(* Logix 5000 project; controller IOL_Sample vendor 1 type 14 code 196 rev 30.11; software revision 30.02; part 5 of 7 *)

           TBEN_L4_8IOL:O.Data[90].9   // IO-Link Port 6 - Output data word 8 (INT bit9)
           TBEN_L4_8IOL:O.Data[90].10   // IO-Link Port 6 - Output data word 8 (INT bit10)
           TBEN_L4_8IOL:O.Data[90].11   // IO-Link Port 6 - Output data word 8 (INT bit11)
           TBEN_L4_8IOL:O.Data[90].12   // IO-Link Port 6 - Output data word 8 (INT bit12)
           TBEN_L4_8IOL:O.Data[90].13   // IO-Link Port 6 - Output data word 8 (INT bit13)
           TBEN_L4_8IOL:O.Data[90].14   // IO-Link Port 6 - Output data word 8 (INT bit14)
           TBEN_L4_8IOL:O.Data[90].15   // IO-Link Port 6 - Output data word 8 (INT bit15)
           TBEN_L4_8IOL:O.Data[91]   // IO-Link Port 6 - Output data word 9
           TBEN_L4_8IOL:O.Data[91].0   // IO-Link Port 6 - Output data word 9 (INT bit0)
           TBEN_L4_8IOL:O.Data[91].1   // IO-Link Port 6 - Output data word 9 (INT bit1)
           TBEN_L4_8IOL:O.Data[91].2   // IO-Link Port 6 - Output data word 9 (INT bit2)
           TBEN_L4_8IOL:O.Data[91].3   // IO-Link Port 6 - Output data word 9 (INT bit3)
           TBEN_L4_8IOL:O.Data[91].4   // IO-Link Port 6 - Output data word 9 (INT bit4)
           TBEN_L4_8IOL:O.Data[91].5   // IO-Link Port 6 - Output data word 9 (INT bit5)
           TBEN_L4_8IOL:O.Data[91].6   // IO-Link Port 6 - Output data word 9 (INT bit6)
           TBEN_L4_8IOL:O.Data[91].7   // IO-Link Port 6 - Output data word 9 (INT bit7)
           TBEN_L4_8IOL:O.Data[91].8   // IO-Link Port 6 - Output data word 9 (INT bit8)
           TBEN_L4_8IOL:O.Data[91].9   // IO-Link Port 6 - Output data word 9 (INT bit9)
           TBEN_L4_8IOL:O.Data[91].10   // IO-Link Port 6 - Output data word 9 (INT bit10)
           TBEN_L4_8IOL:O.Data[91].11   // IO-Link Port 6 - Output data word 9 (INT bit11)
           TBEN_L4_8IOL:O.Data[91].12   // IO-Link Port 6 - Output data word 9 (INT bit12)
           TBEN_L4_8IOL:O.Data[91].13   // IO-Link Port 6 - Output data word 9 (INT bit13)
           TBEN_L4_8IOL:O.Data[91].14   // IO-Link Port 6 - Output data word 9 (INT bit14)
           TBEN_L4_8IOL:O.Data[91].15   // IO-Link Port 6 - Output data word 9 (INT bit15)
           TBEN_L4_8IOL:O.Data[92]   // IO-Link Port 6 - Output data word 10
           TBEN_L4_8IOL:O.Data[92].0   // IO-Link Port 6 - Output data word 10 (INT bit0)
           TBEN_L4_8IOL:O.Data[92].1   // IO-Link Port 6 - Output data word 10 (INT bit1)
           TBEN_L4_8IOL:O.Data[92].2   // IO-Link Port 6 - Output data word 10 (INT bit2)
           TBEN_L4_8IOL:O.Data[92].3   // IO-Link Port 6 - Output data word 10 (INT bit3)
           TBEN_L4_8IOL:O.Data[92].4   // IO-Link Port 6 - Output data word 10 (INT bit4)
           TBEN_L4_8IOL:O.Data[92].5   // IO-Link Port 6 - Output data word 10 (INT bit5)
           TBEN_L4_8IOL:O.Data[92].6   // IO-Link Port 6 - Output data word 10 (INT bit6)
           TBEN_L4_8IOL:O.Data[92].7   // IO-Link Port 6 - Output data word 10 (INT bit7)
           TBEN_L4_8IOL:O.Data[92].8   // IO-Link Port 6 - Output data word 10 (INT bit8)
           TBEN_L4_8IOL:O.Data[92].9   // IO-Link Port 6 - Output data word 10 (INT bit9)
           TBEN_L4_8IOL:O.Data[92].10   // IO-Link Port 6 - Output data word 10 (INT bit10)
           TBEN_L4_8IOL:O.Data[92].11   // IO-Link Port 6 - Output data word 10 (INT bit11)
           TBEN_L4_8IOL:O.Data[92].12   // IO-Link Port 6 - Output data word 10 (INT bit12)
           TBEN_L4_8IOL:O.Data[92].13   // IO-Link Port 6 - Output data word 10 (INT bit13)
           TBEN_L4_8IOL:O.Data[92].14   // IO-Link Port 6 - Output data word 10 (INT bit14)
           TBEN_L4_8IOL:O.Data[92].15   // IO-Link Port 6 - Output data word 10 (INT bit15)
           TBEN_L4_8IOL:O.Data[93]   // IO-Link Port 6 - Output data word 11
           TBEN_L4_8IOL:O.Data[93].0   // IO-Link Port 6 - Output data word 11 (INT bit0)
           TBEN_L4_8IOL:O.Data[93].1   // IO-Link Port 6 - Output data word 11 (INT bit1)
           TBEN_L4_8IOL:O.Data[93].2   // IO-Link Port 6 - Output data word 11 (INT bit2)
           TBEN_L4_8IOL:O.Data[93].3   // IO-Link Port 6 - Output data word 11 (INT bit3)
           TBEN_L4_8IOL:O.Data[93].4   // IO-Link Port 6 - Output data word 11 (INT bit4)
           TBEN_L4_8IOL:O.Data[93].5   // IO-Link Port 6 - Output data word 11 (INT bit5)
           TBEN_L4_8IOL:O.Data[93].6   // IO-Link Port 6 - Output data word 11 (INT bit6)
           TBEN_L4_8IOL:O.Data[93].7   // IO-Link Port 6 - Output data word 11 (INT bit7)
           TBEN_L4_8IOL:O.Data[93].8   // IO-Link Port 6 - Output data word 11 (INT bit8)
           TBEN_L4_8IOL:O.Data[93].9   // IO-Link Port 6 - Output data word 11 (INT bit9)
           TBEN_L4_8IOL:O.Data[93].10   // IO-Link Port 6 - Output data word 11 (INT bit10)
           TBEN_L4_8IOL:O.Data[93].11   // IO-Link Port 6 - Output data word 11 (INT bit11)
           TBEN_L4_8IOL:O.Data[93].12   // IO-Link Port 6 - Output data word 11 (INT bit12)
           TBEN_L4_8IOL:O.Data[93].13   // IO-Link Port 6 - Output data word 11 (INT bit13)
           TBEN_L4_8IOL:O.Data[93].14   // IO-Link Port 6 - Output data word 11 (INT bit14)
           TBEN_L4_8IOL:O.Data[93].15   // IO-Link Port 6 - Output data word 11 (INT bit15)
           TBEN_L4_8IOL:O.Data[94]   // IO-Link Port 6 - Output data word 12
           TBEN_L4_8IOL:O.Data[94].0   // IO-Link Port 6 - Output data word 12 (INT bit0)
           TBEN_L4_8IOL:O.Data[94].1   // IO-Link Port 6 - Output data word 12 (INT bit1)
           TBEN_L4_8IOL:O.Data[94].2   // IO-Link Port 6 - Output data word 12 (INT bit2)
           TBEN_L4_8IOL:O.Data[94].3   // IO-Link Port 6 - Output data word 12 (INT bit3)
           TBEN_L4_8IOL:O.Data[94].4   // IO-Link Port 6 - Output data word 12 (INT bit4)
           TBEN_L4_8IOL:O.Data[94].5   // IO-Link Port 6 - Output data word 12 (INT bit5)
           TBEN_L4_8IOL:O.Data[94].6   // IO-Link Port 6 - Output data word 12 (INT bit6)
           TBEN_L4_8IOL:O.Data[94].7   // IO-Link Port 6 - Output data word 12 (INT bit7)
           TBEN_L4_8IOL:O.Data[94].8   // IO-Link Port 6 - Output data word 12 (INT bit8)
           TBEN_L4_8IOL:O.Data[94].9   // IO-Link Port 6 - Output data word 12 (INT bit9)
           TBEN_L4_8IOL:O.Data[94].10   // IO-Link Port 6 - Output data word 12 (INT bit10)
           TBEN_L4_8IOL:O.Data[94].11   // IO-Link Port 6 - Output data word 12 (INT bit11)
           TBEN_L4_8IOL:O.Data[94].12   // IO-Link Port 6 - Output data word 12 (INT bit12)
           TBEN_L4_8IOL:O.Data[94].13   // IO-Link Port 6 - Output data word 12 (INT bit13)
           TBEN_L4_8IOL:O.Data[94].14   // IO-Link Port 6 - Output data word 12 (INT bit14)
           TBEN_L4_8IOL:O.Data[94].15   // IO-Link Port 6 - Output data word 12 (INT bit15)
           TBEN_L4_8IOL:O.Data[95]   // IO-Link Port 6 - Output data word 13
           TBEN_L4_8IOL:O.Data[95].0   // IO-Link Port 6 - Output data word 13 (INT bit0)
           TBEN_L4_8IOL:O.Data[95].1   // IO-Link Port 6 - Output data word 13 (INT bit1)
           TBEN_L4_8IOL:O.Data[95].2   // IO-Link Port 6 - Output data word 13 (INT bit2)
           TBEN_L4_8IOL:O.Data[95].3   // IO-Link Port 6 - Output data word 13 (INT bit3)
           TBEN_L4_8IOL:O.Data[95].4   // IO-Link Port 6 - Output data word 13 (INT bit4)
           TBEN_L4_8IOL:O.Data[95].5   // IO-Link Port 6 - Output data word 13 (INT bit5)
           TBEN_L4_8IOL:O.Data[95].6   // IO-Link Port 6 - Output data word 13 (INT bit6)
           TBEN_L4_8IOL:O.Data[95].7   // IO-Link Port 6 - Output data word 13 (INT bit7)
           TBEN_L4_8IOL:O.Data[95].8   // IO-Link Port 6 - Output data word 13 (INT bit8)
           TBEN_L4_8IOL:O.Data[95].9   // IO-Link Port 6 - Output data word 13 (INT bit9)
           TBEN_L4_8IOL:O.Data[95].10   // IO-Link Port 6 - Output data word 13 (INT bit10)
           TBEN_L4_8IOL:O.Data[95].11   // IO-Link Port 6 - Output data word 13 (INT bit11)
           TBEN_L4_8IOL:O.Data[95].12   // IO-Link Port 6 - Output data word 13 (INT bit12)
           TBEN_L4_8IOL:O.Data[95].13   // IO-Link Port 6 - Output data word 13 (INT bit13)
           TBEN_L4_8IOL:O.Data[95].14   // IO-Link Port 6 - Output data word 13 (INT bit14)
           TBEN_L4_8IOL:O.Data[95].15   // IO-Link Port 6 - Output data word 13 (INT bit15)
           TBEN_L4_8IOL:O.Data[96]   // IO-Link Port 6 - Output data word 14
           TBEN_L4_8IOL:O.Data[96].0   // IO-Link Port 6 - Output data word 14 (INT bit0)
           TBEN_L4_8IOL:O.Data[96].1   // IO-Link Port 6 - Output data word 14 (INT bit1)
           TBEN_L4_8IOL:O.Data[96].2   // IO-Link Port 6 - Output data word 14 (INT bit2)
           TBEN_L4_8IOL:O.Data[96].3   // IO-Link Port 6 - Output data word 14 (INT bit3)
           TBEN_L4_8IOL:O.Data[96].4   // IO-Link Port 6 - Output data word 14 (INT bit4)
           TBEN_L4_8IOL:O.Data[96].5   // IO-Link Port 6 - Output data word 14 (INT bit5)
           TBEN_L4_8IOL:O.Data[96].6   // IO-Link Port 6 - Output data word 14 (INT bit6)
           TBEN_L4_8IOL:O.Data[96].7   // IO-Link Port 6 - Output data word 14 (INT bit7)
           TBEN_L4_8IOL:O.Data[96].8   // IO-Link Port 6 - Output data word 14 (INT bit8)
           TBEN_L4_8IOL:O.Data[96].9   // IO-Link Port 6 - Output data word 14 (INT bit9)
           TBEN_L4_8IOL:O.Data[96].10   // IO-Link Port 6 - Output data word 14 (INT bit10)
           TBEN_L4_8IOL:O.Data[96].11   // IO-Link Port 6 - Output data word 14 (INT bit11)
           TBEN_L4_8IOL:O.Data[96].12   // IO-Link Port 6 - Output data word 14 (INT bit12)
           TBEN_L4_8IOL:O.Data[96].13   // IO-Link Port 6 - Output data word 14 (INT bit13)
           TBEN_L4_8IOL:O.Data[96].14   // IO-Link Port 6 - Output data word 14 (INT bit14)
           TBEN_L4_8IOL:O.Data[96].15   // IO-Link Port 6 - Output data word 14 (INT bit15)
           TBEN_L4_8IOL:O.Data[97]   // IO-Link Port 6 - Output data word 15
           TBEN_L4_8IOL:O.Data[97].0   // IO-Link Port 6 - Output data word 15 (INT bit0)
           TBEN_L4_8IOL:O.Data[97].1   // IO-Link Port 6 - Output data word 15 (INT bit1)
           TBEN_L4_8IOL:O.Data[97].2   // IO-Link Port 6 - Output data word 15 (INT bit2)
           TBEN_L4_8IOL:O.Data[97].3   // IO-Link Port 6 - Output data word 15 (INT bit3)
           TBEN_L4_8IOL:O.Data[97].4   // IO-Link Port 6 - Output data word 15 (INT bit4)
           TBEN_L4_8IOL:O.Data[97].5   // IO-Link Port 6 - Output data word 15 (INT bit5)
           TBEN_L4_8IOL:O.Data[97].6   // IO-Link Port 6 - Output data word 15 (INT bit6)
           TBEN_L4_8IOL:O.Data[97].7   // IO-Link Port 6 - Output data word 15 (INT bit7)
           TBEN_L4_8IOL:O.Data[97].8   // IO-Link Port 6 - Output data word 15 (INT bit8)
           TBEN_L4_8IOL:O.Data[97].9   // IO-Link Port 6 - Output data word 15 (INT bit9)
           TBEN_L4_8IOL:O.Data[97].10   // IO-Link Port 6 - Output data word 15 (INT bit10)
           TBEN_L4_8IOL:O.Data[97].11   // IO-Link Port 6 - Output data word 15 (INT bit11)
           TBEN_L4_8IOL:O.Data[97].12   // IO-Link Port 6 - Output data word 15 (INT bit12)
           TBEN_L4_8IOL:O.Data[97].13   // IO-Link Port 6 - Output data word 15 (INT bit13)
           TBEN_L4_8IOL:O.Data[97].14   // IO-Link Port 6 - Output data word 15 (INT bit14)
           TBEN_L4_8IOL:O.Data[97].15   // IO-Link Port 6 - Output data word 15 (INT bit15)
           TBEN_L4_8IOL:O.Data[98]   // IO-Link Port 7 - Output data word 0
           TBEN_L4_8IOL:O.Data[98].0   // IO-Link Port 7 - Output data word 0 (INT bit0)
           TBEN_L4_8IOL:O.Data[98].1   // IO-Link Port 7 - Output data word 0 (INT bit1)
           TBEN_L4_8IOL:O.Data[98].2   // IO-Link Port 7 - Output data word 0 (INT bit2)
           TBEN_L4_8IOL:O.Data[98].3   // IO-Link Port 7 - Output data word 0 (INT bit3)
           TBEN_L4_8IOL:O.Data[98].4   // IO-Link Port 7 - Output data word 0 (INT bit4)
           TBEN_L4_8IOL:O.Data[98].5   // IO-Link Port 7 - Output data word 0 (INT bit5)
           TBEN_L4_8IOL:O.Data[98].6   // IO-Link Port 7 - Output data word 0 (INT bit6)
           TBEN_L4_8IOL:O.Data[98].7   // IO-Link Port 7 - Output data word 0 (INT bit7)
           TBEN_L4_8IOL:O.Data[98].8   // IO-Link Port 7 - Output data word 0 (INT bit8)
           TBEN_L4_8IOL:O.Data[98].9   // IO-Link Port 7 - Output data word 0 (INT bit9)
           TBEN_L4_8IOL:O.Data[98].10   // IO-Link Port 7 - Output data word 0 (INT bit10)
           TBEN_L4_8IOL:O.Data[98].11   // IO-Link Port 7 - Output data word 0 (INT bit11)
           TBEN_L4_8IOL:O.Data[98].12   // IO-Link Port 7 - Output data word 0 (INT bit12)
           TBEN_L4_8IOL:O.Data[98].13   // IO-Link Port 7 - Output data word 0 (INT bit13)
           TBEN_L4_8IOL:O.Data[98].14   // IO-Link Port 7 - Output data word 0 (INT bit14)
           TBEN_L4_8IOL:O.Data[98].15   // IO-Link Port 7 - Output data word 0 (INT bit15)
           TBEN_L4_8IOL:O.Data[99]   // IO-Link Port 7 - Output data word 1
           TBEN_L4_8IOL:O.Data[99].0   // IO-Link Port 7 - Output data word 1 (INT bit0)
           TBEN_L4_8IOL:O.Data[99].1   // IO-Link Port 7 - Output data word 1 (INT bit1)
           TBEN_L4_8IOL:O.Data[99].2   // IO-Link Port 7 - Output data word 1 (INT bit2)
           TBEN_L4_8IOL:O.Data[99].3   // IO-Link Port 7 - Output data word 1 (INT bit3)
           TBEN_L4_8IOL:O.Data[99].4   // IO-Link Port 7 - Output data word 1 (INT bit4)
           TBEN_L4_8IOL:O.Data[99].5   // IO-Link Port 7 - Output data word 1 (INT bit5)
           TBEN_L4_8IOL:O.Data[99].6   // IO-Link Port 7 - Output data word 1 (INT bit6)
           TBEN_L4_8IOL:O.Data[99].7   // IO-Link Port 7 - Output data word 1 (INT bit7)
           TBEN_L4_8IOL:O.Data[99].8   // IO-Link Port 7 - Output data word 1 (INT bit8)
           TBEN_L4_8IOL:O.Data[99].9   // IO-Link Port 7 - Output data word 1 (INT bit9)
           TBEN_L4_8IOL:O.Data[99].10   // IO-Link Port 7 - Output data word 1 (INT bit10)
           TBEN_L4_8IOL:O.Data[99].11   // IO-Link Port 7 - Output data word 1 (INT bit11)
           TBEN_L4_8IOL:O.Data[99].12   // IO-Link Port 7 - Output data word 1 (INT bit12)
           TBEN_L4_8IOL:O.Data[99].13   // IO-Link Port 7 - Output data word 1 (INT bit13)
           TBEN_L4_8IOL:O.Data[99].14   // IO-Link Port 7 - Output data word 1 (INT bit14)
           TBEN_L4_8IOL:O.Data[99].15   // IO-Link Port 7 - Output data word 1 (INT bit15)
           TBEN_L4_8IOL:O.Data[100]   // IO-Link Port 7 - Output data word 2
           TBEN_L4_8IOL:O.Data[100].0   // IO-Link Port 7 - Output data word 2 (INT bit0)
           TBEN_L4_8IOL:O.Data[100].1   // IO-Link Port 7 - Output data word 2 (INT bit1)
           TBEN_L4_8IOL:O.Data[100].2   // IO-Link Port 7 - Output data word 2 (INT bit2)
           TBEN_L4_8IOL:O.Data[100].3   // IO-Link Port 7 - Output data word 2 (INT bit3)
           TBEN_L4_8IOL:O.Data[100].4   // IO-Link Port 7 - Output data word 2 (INT bit4)
           TBEN_L4_8IOL:O.Data[100].5   // IO-Link Port 7 - Output data word 2 (INT bit5)
           TBEN_L4_8IOL:O.Data[100].6   // IO-Link Port 7 - Output data word 2 (INT bit6)
           TBEN_L4_8IOL:O.Data[100].7   // IO-Link Port 7 - Output data word 2 (INT bit7)
           TBEN_L4_8IOL:O.Data[100].8   // IO-Link Port 7 - Output data word 2 (INT bit8)
           TBEN_L4_8IOL:O.Data[100].9   // IO-Link Port 7 - Output data word 2 (INT bit9)
           TBEN_L4_8IOL:O.Data[100].10   // IO-Link Port 7 - Output data word 2 (INT bit10)
           TBEN_L4_8IOL:O.Data[100].11   // IO-Link Port 7 - Output data word 2 (INT bit11)
           TBEN_L4_8IOL:O.Data[100].12   // IO-Link Port 7 - Output data word 2 (INT bit12)
           TBEN_L4_8IOL:O.Data[100].13   // IO-Link Port 7 - Output data word 2 (INT bit13)
           TBEN_L4_8IOL:O.Data[100].14   // IO-Link Port 7 - Output data word 2 (INT bit14)
           TBEN_L4_8IOL:O.Data[100].15   // IO-Link Port 7 - Output data word 2 (INT bit15)
           TBEN_L4_8IOL:O.Data[101]   // IO-Link Port 7 - Output data word 3
           TBEN_L4_8IOL:O.Data[101].0   // IO-Link Port 7 - Output data word 3 (INT bit0)
           TBEN_L4_8IOL:O.Data[101].1   // IO-Link Port 7 - Output data word 3 (INT bit1)
           TBEN_L4_8IOL:O.Data[101].2   // IO-Link Port 7 - Output data word 3 (INT bit2)
           TBEN_L4_8IOL:O.Data[101].3   // IO-Link Port 7 - Output data word 3 (INT bit3)
           TBEN_L4_8IOL:O.Data[101].4   // IO-Link Port 7 - Output data word 3 (INT bit4)
           TBEN_L4_8IOL:O.Data[101].5   // IO-Link Port 7 - Output data word 3 (INT bit5)
           TBEN_L4_8IOL:O.Data[101].6   // IO-Link Port 7 - Output data word 3 (INT bit6)
           TBEN_L4_8IOL:O.Data[101].7   // IO-Link Port 7 - Output data word 3 (INT bit7)
           TBEN_L4_8IOL:O.Data[101].8   // IO-Link Port 7 - Output data word 3 (INT bit8)
           TBEN_L4_8IOL:O.Data[101].9   // IO-Link Port 7 - Output data word 3 (INT bit9)
           TBEN_L4_8IOL:O.Data[101].10   // IO-Link Port 7 - Output data word 3 (INT bit10)
           TBEN_L4_8IOL:O.Data[101].11   // IO-Link Port 7 - Output data word 3 (INT bit11)
           TBEN_L4_8IOL:O.Data[101].12   // IO-Link Port 7 - Output data word 3 (INT bit12)
           TBEN_L4_8IOL:O.Data[101].13   // IO-Link Port 7 - Output data word 3 (INT bit13)
           TBEN_L4_8IOL:O.Data[101].14   // IO-Link Port 7 - Output data word 3 (INT bit14)
           TBEN_L4_8IOL:O.Data[101].15   // IO-Link Port 7 - Output data word 3 (INT bit15)
           TBEN_L4_8IOL:O.Data[102]   // IO-Link Port 7 - Output data word 4
           TBEN_L4_8IOL:O.Data[102].0   // IO-Link Port 7 - Output data word 4 (INT bit0)
           TBEN_L4_8IOL:O.Data[102].1   // IO-Link Port 7 - Output data word 4 (INT bit1)
           TBEN_L4_8IOL:O.Data[102].2   // IO-Link Port 7 - Output data word 4 (INT bit2)
           TBEN_L4_8IOL:O.Data[102].3   // IO-Link Port 7 - Output data word 4 (INT bit3)
           TBEN_L4_8IOL:O.Data[102].4   // IO-Link Port 7 - Output data word 4 (INT bit4)
           TBEN_L4_8IOL:O.Data[102].5   // IO-Link Port 7 - Output data word 4 (INT bit5)
           TBEN_L4_8IOL:O.Data[102].6   // IO-Link Port 7 - Output data word 4 (INT bit6)
           TBEN_L4_8IOL:O.Data[102].7   // IO-Link Port 7 - Output data word 4 (INT bit7)
           TBEN_L4_8IOL:O.Data[102].8   // IO-Link Port 7 - Output data word 4 (INT bit8)
           TBEN_L4_8IOL:O.Data[102].9   // IO-Link Port 7 - Output data word 4 (INT bit9)
           TBEN_L4_8IOL:O.Data[102].10   // IO-Link Port 7 - Output data word 4 (INT bit10)
           TBEN_L4_8IOL:O.Data[102].11   // IO-Link Port 7 - Output data word 4 (INT bit11)
           TBEN_L4_8IOL:O.Data[102].12   // IO-Link Port 7 - Output data word 4 (INT bit12)
           TBEN_L4_8IOL:O.Data[102].13   // IO-Link Port 7 - Output data word 4 (INT bit13)
           TBEN_L4_8IOL:O.Data[102].14   // IO-Link Port 7 - Output data word 4 (INT bit14)
           TBEN_L4_8IOL:O.Data[102].15   // IO-Link Port 7 - Output data word 4 (INT bit15)
           TBEN_L4_8IOL:O.Data[103]   // IO-Link Port 7 - Output data word 5
           TBEN_L4_8IOL:O.Data[103].0   // IO-Link Port 7 - Output data word 5 (INT bit0)
           TBEN_L4_8IOL:O.Data[103].1   // IO-Link Port 7 - Output data word 5 (INT bit1)
           TBEN_L4_8IOL:O.Data[103].2   // IO-Link Port 7 - Output data word 5 (INT bit2)
           TBEN_L4_8IOL:O.Data[103].3   // IO-Link Port 7 - Output data word 5 (INT bit3)
           TBEN_L4_8IOL:O.Data[103].4   // IO-Link Port 7 - Output data word 5 (INT bit4)
           TBEN_L4_8IOL:O.Data[103].5   // IO-Link Port 7 - Output data word 5 (INT bit5)
           TBEN_L4_8IOL:O.Data[103].6   // IO-Link Port 7 - Output data word 5 (INT bit6)
           TBEN_L4_8IOL:O.Data[103].7   // IO-Link Port 7 - Output data word 5 (INT bit7)
           TBEN_L4_8IOL:O.Data[103].8   // IO-Link Port 7 - Output data word 5 (INT bit8)
           TBEN_L4_8IOL:O.Data[103].9   // IO-Link Port 7 - Output data word 5 (INT bit9)
           TBEN_L4_8IOL:O.Data[103].10   // IO-Link Port 7 - Output data word 5 (INT bit10)
           TBEN_L4_8IOL:O.Data[103].11   // IO-Link Port 7 - Output data word 5 (INT bit11)
           TBEN_L4_8IOL:O.Data[103].12   // IO-Link Port 7 - Output data word 5 (INT bit12)
           TBEN_L4_8IOL:O.Data[103].13   // IO-Link Port 7 - Output data word 5 (INT bit13)
           TBEN_L4_8IOL:O.Data[103].14   // IO-Link Port 7 - Output data word 5 (INT bit14)
           TBEN_L4_8IOL:O.Data[103].15   // IO-Link Port 7 - Output data word 5 (INT bit15)
           TBEN_L4_8IOL:O.Data[104]   // IO-Link Port 7 - Output data word 6
           TBEN_L4_8IOL:O.Data[104].0   // IO-Link Port 7 - Output data word 6 (INT bit0)
           TBEN_L4_8IOL:O.Data[104].1   // IO-Link Port 7 - Output data word 6 (INT bit1)
           TBEN_L4_8IOL:O.Data[104].2   // IO-Link Port 7 - Output data word 6 (INT bit2)
           TBEN_L4_8IOL:O.Data[104].3   // IO-Link Port 7 - Output data word 6 (INT bit3)
           TBEN_L4_8IOL:O.Data[104].4   // IO-Link Port 7 - Output data word 6 (INT bit4)
           TBEN_L4_8IOL:O.Data[104].5   // IO-Link Port 7 - Output data word 6 (INT bit5)
           TBEN_L4_8IOL:O.Data[104].6   // IO-Link Port 7 - Output data word 6 (INT bit6)
           TBEN_L4_8IOL:O.Data[104].7   // IO-Link Port 7 - Output data word 6 (INT bit7)
           TBEN_L4_8IOL:O.Data[104].8   // IO-Link Port 7 - Output data word 6 (INT bit8)
           TBEN_L4_8IOL:O.Data[104].9   // IO-Link Port 7 - Output data word 6 (INT bit9)
           TBEN_L4_8IOL:O.Data[104].10   // IO-Link Port 7 - Output data word 6 (INT bit10)
           TBEN_L4_8IOL:O.Data[104].11   // IO-Link Port 7 - Output data word 6 (INT bit11)
           TBEN_L4_8IOL:O.Data[104].12   // IO-Link Port 7 - Output data word 6 (INT bit12)
           TBEN_L4_8IOL:O.Data[104].13   // IO-Link Port 7 - Output data word 6 (INT bit13)
           TBEN_L4_8IOL:O.Data[104].14   // IO-Link Port 7 - Output data word 6 (INT bit14)
           TBEN_L4_8IOL:O.Data[104].15   // IO-Link Port 7 - Output data word 6 (INT bit15)
           TBEN_L4_8IOL:O.Data[105]   // IO-Link Port 7 - Output data word 7
           TBEN_L4_8IOL:O.Data[105].0   // IO-Link Port 7 - Output data word 7 (INT bit0)
           TBEN_L4_8IOL:O.Data[105].1   // IO-Link Port 7 - Output data word 7 (INT bit1)
           TBEN_L4_8IOL:O.Data[105].2   // IO-Link Port 7 - Output data word 7 (INT bit2)
           TBEN_L4_8IOL:O.Data[105].3   // IO-Link Port 7 - Output data word 7 (INT bit3)
           TBEN_L4_8IOL:O.Data[105].4   // IO-Link Port 7 - Output data word 7 (INT bit4)
           TBEN_L4_8IOL:O.Data[105].5   // IO-Link Port 7 - Output data word 7 (INT bit5)
           TBEN_L4_8IOL:O.Data[105].6   // IO-Link Port 7 - Output data word 7 (INT bit6)
           TBEN_L4_8IOL:O.Data[105].7   // IO-Link Port 7 - Output data word 7 (INT bit7)
           TBEN_L4_8IOL:O.Data[105].8   // IO-Link Port 7 - Output data word 7 (INT bit8)
           TBEN_L4_8IOL:O.Data[105].9   // IO-Link Port 7 - Output data word 7 (INT bit9)
           TBEN_L4_8IOL:O.Data[105].10   // IO-Link Port 7 - Output data word 7 (INT bit10)
           TBEN_L4_8IOL:O.Data[105].11   // IO-Link Port 7 - Output data word 7 (INT bit11)
           TBEN_L4_8IOL:O.Data[105].12   // IO-Link Port 7 - Output data word 7 (INT bit12)
           TBEN_L4_8IOL:O.Data[105].13   // IO-Link Port 7 - Output data word 7 (INT bit13)
           TBEN_L4_8IOL:O.Data[105].14   // IO-Link Port 7 - Output data word 7 (INT bit14)
           TBEN_L4_8IOL:O.Data[105].15   // IO-Link Port 7 - Output data word 7 (INT bit15)
           TBEN_L4_8IOL:O.Data[106]   // IO-Link Port 7 - Output data word 8
           TBEN_L4_8IOL:O.Data[106].0   // IO-Link Port 7 - Output data word 8 (INT bit0)
           TBEN_L4_8IOL:O.Data[106].1   // IO-Link Port 7 - Output data word 8 (INT bit1)
           TBEN_L4_8IOL:O.Data[106].2   // IO-Link Port 7 - Output data word 8 (INT bit2)
           TBEN_L4_8IOL:O.Data[106].3   // IO-Link Port 7 - Output data word 8 (INT bit3)
           TBEN_L4_8IOL:O.Data[106].4   // IO-Link Port 7 - Output data word 8 (INT bit4)
           TBEN_L4_8IOL:O.Data[106].5   // IO-Link Port 7 - Output data word 8 (INT bit5)
           TBEN_L4_8IOL:O.Data[106].6   // IO-Link Port 7 - Output data word 8 (INT bit6)
           TBEN_L4_8IOL:O.Data[106].7   // IO-Link Port 7 - Output data word 8 (INT bit7)
           TBEN_L4_8IOL:O.Data[106].8   // IO-Link Port 7 - Output data word 8 (INT bit8)
           TBEN_L4_8IOL:O.Data[106].9   // IO-Link Port 7 - Output data word 8 (INT bit9)
           TBEN_L4_8IOL:O.Data[106].10   // IO-Link Port 7 - Output data word 8 (INT bit10)
           TBEN_L4_8IOL:O.Data[106].11   // IO-Link Port 7 - Output data word 8 (INT bit11)
           TBEN_L4_8IOL:O.Data[106].12   // IO-Link Port 7 - Output data word 8 (INT bit12)
           TBEN_L4_8IOL:O.Data[106].13   // IO-Link Port 7 - Output data word 8 (INT bit13)
           TBEN_L4_8IOL:O.Data[106].14   // IO-Link Port 7 - Output data word 8 (INT bit14)
           TBEN_L4_8IOL:O.Data[106].15   // IO-Link Port 7 - Output data word 8 (INT bit15)
           TBEN_L4_8IOL:O.Data[107]   // IO-Link Port 7 - Output data word 9
           TBEN_L4_8IOL:O.Data[107].0   // IO-Link Port 7 - Output data word 9 (INT bit0)
           TBEN_L4_8IOL:O.Data[107].1   // IO-Link Port 7 - Output data word 9 (INT bit1)
           TBEN_L4_8IOL:O.Data[107].2   // IO-Link Port 7 - Output data word 9 (INT bit2)
           TBEN_L4_8IOL:O.Data[107].3   // IO-Link Port 7 - Output data word 9 (INT bit3)
           TBEN_L4_8IOL:O.Data[107].4   // IO-Link Port 7 - Output data word 9 (INT bit4)
           TBEN_L4_8IOL:O.Data[107].5   // IO-Link Port 7 - Output data word 9 (INT bit5)
           TBEN_L4_8IOL:O.Data[107].6   // IO-Link Port 7 - Output data word 9 (INT bit6)
           TBEN_L4_8IOL:O.Data[107].7   // IO-Link Port 7 - Output data word 9 (INT bit7)
           TBEN_L4_8IOL:O.Data[107].8   // IO-Link Port 7 - Output data word 9 (INT bit8)
           TBEN_L4_8IOL:O.Data[107].9   // IO-Link Port 7 - Output data word 9 (INT bit9)
           TBEN_L4_8IOL:O.Data[107].10   // IO-Link Port 7 - Output data word 9 (INT bit10)
           TBEN_L4_8IOL:O.Data[107].11   // IO-Link Port 7 - Output data word 9 (INT bit11)
           TBEN_L4_8IOL:O.Data[107].12   // IO-Link Port 7 - Output data word 9 (INT bit12)
           TBEN_L4_8IOL:O.Data[107].13   // IO-Link Port 7 - Output data word 9 (INT bit13)
           TBEN_L4_8IOL:O.Data[107].14   // IO-Link Port 7 - Output data word 9 (INT bit14)
           TBEN_L4_8IOL:O.Data[107].15   // IO-Link Port 7 - Output data word 9 (INT bit15)
           TBEN_L4_8IOL:O.Data[108]   // IO-Link Port 7 - Output data word 10
           TBEN_L4_8IOL:O.Data[108].0   // IO-Link Port 7 - Output data word 10 (INT bit0)
           TBEN_L4_8IOL:O.Data[108].1   // IO-Link Port 7 - Output data word 10 (INT bit1)
           TBEN_L4_8IOL:O.Data[108].2   // IO-Link Port 7 - Output data word 10 (INT bit2)
           TBEN_L4_8IOL:O.Data[108].3   // IO-Link Port 7 - Output data word 10 (INT bit3)
           TBEN_L4_8IOL:O.Data[108].4   // IO-Link Port 7 - Output data word 10 (INT bit4)
           TBEN_L4_8IOL:O.Data[108].5   // IO-Link Port 7 - Output data word 10 (INT bit5)
           TBEN_L4_8IOL:O.Data[108].6   // IO-Link Port 7 - Output data word 10 (INT bit6)
           TBEN_L4_8IOL:O.Data[108].7   // IO-Link Port 7 - Output data word 10 (INT bit7)
           TBEN_L4_8IOL:O.Data[108].8   // IO-Link Port 7 - Output data word 10 (INT bit8)
           TBEN_L4_8IOL:O.Data[108].9   // IO-Link Port 7 - Output data word 10 (INT bit9)
           TBEN_L4_8IOL:O.Data[108].10   // IO-Link Port 7 - Output data word 10 (INT bit10)
           TBEN_L4_8IOL:O.Data[108].11   // IO-Link Port 7 - Output data word 10 (INT bit11)
           TBEN_L4_8IOL:O.Data[108].12   // IO-Link Port 7 - Output data word 10 (INT bit12)
           TBEN_L4_8IOL:O.Data[108].13   // IO-Link Port 7 - Output data word 10 (INT bit13)
           TBEN_L4_8IOL:O.Data[108].14   // IO-Link Port 7 - Output data word 10 (INT bit14)
           TBEN_L4_8IOL:O.Data[108].15   // IO-Link Port 7 - Output data word 10 (INT bit15)
           TBEN_L4_8IOL:O.Data[109]   // IO-Link Port 7 - Output data word 11
           TBEN_L4_8IOL:O.Data[109].0   // IO-Link Port 7 - Output data word 11 (INT bit0)
           TBEN_L4_8IOL:O.Data[109].1   // IO-Link Port 7 - Output data word 11 (INT bit1)
           TBEN_L4_8IOL:O.Data[109].2   // IO-Link Port 7 - Output data word 11 (INT bit2)
           TBEN_L4_8IOL:O.Data[109].3   // IO-Link Port 7 - Output data word 11 (INT bit3)
           TBEN_L4_8IOL:O.Data[109].4   // IO-Link Port 7 - Output data word 11 (INT bit4)
           TBEN_L4_8IOL:O.Data[109].5   // IO-Link Port 7 - Output data word 11 (INT bit5)
           TBEN_L4_8IOL:O.Data[109].6   // IO-Link Port 7 - Output data word 11 (INT bit6)
           TBEN_L4_8IOL:O.Data[109].7   // IO-Link Port 7 - Output data word 11 (INT bit7)
           TBEN_L4_8IOL:O.Data[109].8   // IO-Link Port 7 - Output data word 11 (INT bit8)
           TBEN_L4_8IOL:O.Data[109].9   // IO-Link Port 7 - Output data word 11 (INT bit9)
           TBEN_L4_8IOL:O.Data[109].10   // IO-Link Port 7 - Output data word 11 (INT bit10)
           TBEN_L4_8IOL:O.Data[109].11   // IO-Link Port 7 - Output data word 11 (INT bit11)
           TBEN_L4_8IOL:O.Data[109].12   // IO-Link Port 7 - Output data word 11 (INT bit12)
           TBEN_L4_8IOL:O.Data[109].13   // IO-Link Port 7 - Output data word 11 (INT bit13)
           TBEN_L4_8IOL:O.Data[109].14   // IO-Link Port 7 - Output data word 11 (INT bit14)
           TBEN_L4_8IOL:O.Data[109].15   // IO-Link Port 7 - Output data word 11 (INT bit15)
           TBEN_L4_8IOL:O.Data[110]   // IO-Link Port 7 - Output data word 12
           TBEN_L4_8IOL:O.Data[110].0   // IO-Link Port 7 - Output data word 12 (INT bit0)
           TBEN_L4_8IOL:O.Data[110].1   // IO-Link Port 7 - Output data word 12 (INT bit1)
           TBEN_L4_8IOL:O.Data[110].2   // IO-Link Port 7 - Output data word 12 (INT bit2)
           TBEN_L4_8IOL:O.Data[110].3   // IO-Link Port 7 - Output data word 12 (INT bit3)
           TBEN_L4_8IOL:O.Data[110].4   // IO-Link Port 7 - Output data word 12 (INT bit4)
           TBEN_L4_8IOL:O.Data[110].5   // IO-Link Port 7 - Output data word 12 (INT bit5)
           TBEN_L4_8IOL:O.Data[110].6   // IO-Link Port 7 - Output data word 12 (INT bit6)
           TBEN_L4_8IOL:O.Data[110].7   // IO-Link Port 7 - Output data word 12 (INT bit7)
           TBEN_L4_8IOL:O.Data[110].8   // IO-Link Port 7 - Output data word 12 (INT bit8)
           TBEN_L4_8IOL:O.Data[110].9   // IO-Link Port 7 - Output data word 12 (INT bit9)
           TBEN_L4_8IOL:O.Data[110].10   // IO-Link Port 7 - Output data word 12 (INT bit10)
           TBEN_L4_8IOL:O.Data[110].11   // IO-Link Port 7 - Output data word 12 (INT bit11)
           TBEN_L4_8IOL:O.Data[110].12   // IO-Link Port 7 - Output data word 12 (INT bit12)
           TBEN_L4_8IOL:O.Data[110].13   // IO-Link Port 7 - Output data word 12 (INT bit13)
           TBEN_L4_8IOL:O.Data[110].14   // IO-Link Port 7 - Output data word 12 (INT bit14)
           TBEN_L4_8IOL:O.Data[110].15   // IO-Link Port 7 - Output data word 12 (INT bit15)
           TBEN_L4_8IOL:O.Data[111]   // IO-Link Port 7 - Output data word 13
           TBEN_L4_8IOL:O.Data[111].0   // IO-Link Port 7 - Output data word 13 (INT bit0)
           TBEN_L4_8IOL:O.Data[111].1   // IO-Link Port 7 - Output data word 13 (INT bit1)
           TBEN_L4_8IOL:O.Data[111].2   // IO-Link Port 7 - Output data word 13 (INT bit2)
           TBEN_L4_8IOL:O.Data[111].3   // IO-Link Port 7 - Output data word 13 (INT bit3)
           TBEN_L4_8IOL:O.Data[111].4   // IO-Link Port 7 - Output data word 13 (INT bit4)
           TBEN_L4_8IOL:O.Data[111].5   // IO-Link Port 7 - Output data word 13 (INT bit5)
           TBEN_L4_8IOL:O.Data[111].6   // IO-Link Port 7 - Output data word 13 (INT bit6)
           TBEN_L4_8IOL:O.Data[111].7   // IO-Link Port 7 - Output data word 13 (INT bit7)
           TBEN_L4_8IOL:O.Data[111].8   // IO-Link Port 7 - Output data word 13 (INT bit8)
           TBEN_L4_8IOL:O.Data[111].9   // IO-Link Port 7 - Output data word 13 (INT bit9)
           TBEN_L4_8IOL:O.Data[111].10   // IO-Link Port 7 - Output data word 13 (INT bit10)
           TBEN_L4_8IOL:O.Data[111].11   // IO-Link Port 7 - Output data word 13 (INT bit11)
           TBEN_L4_8IOL:O.Data[111].12   // IO-Link Port 7 - Output data word 13 (INT bit12)
           TBEN_L4_8IOL:O.Data[111].13   // IO-Link Port 7 - Output data word 13 (INT bit13)
           TBEN_L4_8IOL:O.Data[111].14   // IO-Link Port 7 - Output data word 13 (INT bit14)
           TBEN_L4_8IOL:O.Data[111].15   // IO-Link Port 7 - Output data word 13 (INT bit15)
           TBEN_L4_8IOL:O.Data[112]   // IO-Link Port 7 - Output data word 14
           TBEN_L4_8IOL:O.Data[112].0   // IO-Link Port 7 - Output data word 14 (INT bit0)
           TBEN_L4_8IOL:O.Data[112].1   // IO-Link Port 7 - Output data word 14 (INT bit1)
           TBEN_L4_8IOL:O.Data[112].2   // IO-Link Port 7 - Output data word 14 (INT bit2)
           TBEN_L4_8IOL:O.Data[112].3   // IO-Link Port 7 - Output data word 14 (INT bit3)
           TBEN_L4_8IOL:O.Data[112].4   // IO-Link Port 7 - Output data word 14 (INT bit4)
           TBEN_L4_8IOL:O.Data[112].5   // IO-Link Port 7 - Output data word 14 (INT bit5)
           TBEN_L4_8IOL:O.Data[112].6   // IO-Link Port 7 - Output data word 14 (INT bit6)
           TBEN_L4_8IOL:O.Data[112].7   // IO-Link Port 7 - Output data word 14 (INT bit7)
           TBEN_L4_8IOL:O.Data[112].8   // IO-Link Port 7 - Output data word 14 (INT bit8)
           TBEN_L4_8IOL:O.Data[112].9   // IO-Link Port 7 - Output data word 14 (INT bit9)
           TBEN_L4_8IOL:O.Data[112].10   // IO-Link Port 7 - Output data word 14 (INT bit10)
           TBEN_L4_8IOL:O.Data[112].11   // IO-Link Port 7 - Output data word 14 (INT bit11)
           TBEN_L4_8IOL:O.Data[112].12   // IO-Link Port 7 - Output data word 14 (INT bit12)
           TBEN_L4_8IOL:O.Data[112].13   // IO-Link Port 7 - Output data word 14 (INT bit13)
           TBEN_L4_8IOL:O.Data[112].14   // IO-Link Port 7 - Output data word 14 (INT bit14)
           TBEN_L4_8IOL:O.Data[112].15   // IO-Link Port 7 - Output data word 14 (INT bit15)
           TBEN_L4_8IOL:O.Data[113]   // IO-Link Port 7 - Output data word 15
           TBEN_L4_8IOL:O.Data[113].0   // IO-Link Port 7 - Output data word 15 (INT bit0)
           TBEN_L4_8IOL:O.Data[113].1   // IO-Link Port 7 - Output data word 15 (INT bit1)
           TBEN_L4_8IOL:O.Data[113].2   // IO-Link Port 7 - Output data word 15 (INT bit2)
           TBEN_L4_8IOL:O.Data[113].3   // IO-Link Port 7 - Output data word 15 (INT bit3)
           TBEN_L4_8IOL:O.Data[113].4   // IO-Link Port 7 - Output data word 15 (INT bit4)
           TBEN_L4_8IOL:O.Data[113].5   // IO-Link Port 7 - Output data word 15 (INT bit5)
           TBEN_L4_8IOL:O.Data[113].6   // IO-Link Port 7 - Output data word 15 (INT bit6)
           TBEN_L4_8IOL:O.Data[113].7   // IO-Link Port 7 - Output data word 15 (INT bit7)
           TBEN_L4_8IOL:O.Data[113].8   // IO-Link Port 7 - Output data word 15 (INT bit8)
           TBEN_L4_8IOL:O.Data[113].9   // IO-Link Port 7 - Output data word 15 (INT bit9)
           TBEN_L4_8IOL:O.Data[113].10   // IO-Link Port 7 - Output data word 15 (INT bit10)
           TBEN_L4_8IOL:O.Data[113].11   // IO-Link Port 7 - Output data word 15 (INT bit11)
           TBEN_L4_8IOL:O.Data[113].12   // IO-Link Port 7 - Output data word 15 (INT bit12)
           TBEN_L4_8IOL:O.Data[113].13   // IO-Link Port 7 - Output data word 15 (INT bit13)
           TBEN_L4_8IOL:O.Data[113].14   // IO-Link Port 7 - Output data word 15 (INT bit14)
           TBEN_L4_8IOL:O.Data[113].15   // IO-Link Port 7 - Output data word 15 (INT bit15)
           TBEN_L4_8IOL:O.Data[114]   // IO-Link Port 8 - Output data word 0
           TBEN_L4_8IOL:O.Data[114].0   // IO-Link Port 8 - Output data word 0 (INT bit0)
           TBEN_L4_8IOL:O.Data[114].1   // IO-Link Port 8 - Output data word 0 (INT bit1)
           TBEN_L4_8IOL:O.Data[114].2   // IO-Link Port 8 - Output data word 0 (INT bit2)
           TBEN_L4_8IOL:O.Data[114].3   // IO-Link Port 8 - Output data word 0 (INT bit3)
           TBEN_L4_8IOL:O.Data[114].4   // IO-Link Port 8 - Output data word 0 (INT bit4)
           TBEN_L4_8IOL:O.Data[114].5   // IO-Link Port 8 - Output data word 0 (INT bit5)
           TBEN_L4_8IOL:O.Data[114].6   // IO-Link Port 8 - Output data word 0 (INT bit6)
           TBEN_L4_8IOL:O.Data[114].7   // IO-Link Port 8 - Output data word 0 (INT bit7)
           TBEN_L4_8IOL:O.Data[114].8   // IO-Link Port 8 - Output data word 0 (INT bit8)
           TBEN_L4_8IOL:O.Data[114].9   // IO-Link Port 8 - Output data word 0 (INT bit9)
           TBEN_L4_8IOL:O.Data[114].10   // IO-Link Port 8 - Output data word 0 (INT bit10)
           TBEN_L4_8IOL:O.Data[114].11   // IO-Link Port 8 - Output data word 0 (INT bit11)
           TBEN_L4_8IOL:O.Data[114].12   // IO-Link Port 8 - Output data word 0 (INT bit12)
           TBEN_L4_8IOL:O.Data[114].13   // IO-Link Port 8 - Output data word 0 (INT bit13)
           TBEN_L4_8IOL:O.Data[114].14   // IO-Link Port 8 - Output data word 0 (INT bit14)
           TBEN_L4_8IOL:O.Data[114].15   // IO-Link Port 8 - Output data word 0 (INT bit15)
           TBEN_L4_8IOL:O.Data[115]   // IO-Link Port 8 - Output data word 1
           TBEN_L4_8IOL:O.Data[115].0   // IO-Link Port 8 - Output data word 1 (INT bit0)
           TBEN_L4_8IOL:O.Data[115].1   // IO-Link Port 8 - Output data word 1 (INT bit1)
           TBEN_L4_8IOL:O.Data[115].2   // IO-Link Port 8 - Output data word 1 (INT bit2)
           TBEN_L4_8IOL:O.Data[115].3   // IO-Link Port 8 - Output data word 1 (INT bit3)
           TBEN_L4_8IOL:O.Data[115].4   // IO-Link Port 8 - Output data word 1 (INT bit4)
           TBEN_L4_8IOL:O.Data[115].5   // IO-Link Port 8 - Output data word 1 (INT bit5)
           TBEN_L4_8IOL:O.Data[115].6   // IO-Link Port 8 - Output data word 1 (INT bit6)
           TBEN_L4_8IOL:O.Data[115].7   // IO-Link Port 8 - Output data word 1 (INT bit7)
           TBEN_L4_8IOL:O.Data[115].8   // IO-Link Port 8 - Output data word 1 (INT bit8)
           TBEN_L4_8IOL:O.Data[115].9   // IO-Link Port 8 - Output data word 1 (INT bit9)
           TBEN_L4_8IOL:O.Data[115].10   // IO-Link Port 8 - Output data word 1 (INT bit10)
           TBEN_L4_8IOL:O.Data[115].11   // IO-Link Port 8 - Output data word 1 (INT bit11)
           TBEN_L4_8IOL:O.Data[115].12   // IO-Link Port 8 - Output data word 1 (INT bit12)
           TBEN_L4_8IOL:O.Data[115].13   // IO-Link Port 8 - Output data word 1 (INT bit13)
           TBEN_L4_8IOL:O.Data[115].14   // IO-Link Port 8 - Output data word 1 (INT bit14)
           TBEN_L4_8IOL:O.Data[115].15   // IO-Link Port 8 - Output data word 1 (INT bit15)
           TBEN_L4_8IOL:O.Data[116]   // IO-Link Port 8 - Output data word 2
           TBEN_L4_8IOL:O.Data[116].0   // IO-Link Port 8 - Output data word 2 (INT bit0)
           TBEN_L4_8IOL:O.Data[116].1   // IO-Link Port 8 - Output data word 2 (INT bit1)
           TBEN_L4_8IOL:O.Data[116].2   // IO-Link Port 8 - Output data word 2 (INT bit2)
           TBEN_L4_8IOL:O.Data[116].3   // IO-Link Port 8 - Output data word 2 (INT bit3)
           TBEN_L4_8IOL:O.Data[116].4   // IO-Link Port 8 - Output data word 2 (INT bit4)
           TBEN_L4_8IOL:O.Data[116].5   // IO-Link Port 8 - Output data word 2 (INT bit5)
           TBEN_L4_8IOL:O.Data[116].6   // IO-Link Port 8 - Output data word 2 (INT bit6)
           TBEN_L4_8IOL:O.Data[116].7   // IO-Link Port 8 - Output data word 2 (INT bit7)
           TBEN_L4_8IOL:O.Data[116].8   // IO-Link Port 8 - Output data word 2 (INT bit8)
           TBEN_L4_8IOL:O.Data[116].9   // IO-Link Port 8 - Output data word 2 (INT bit9)
           TBEN_L4_8IOL:O.Data[116].10   // IO-Link Port 8 - Output data word 2 (INT bit10)
           TBEN_L4_8IOL:O.Data[116].11   // IO-Link Port 8 - Output data word 2 (INT bit11)
           TBEN_L4_8IOL:O.Data[116].12   // IO-Link Port 8 - Output data word 2 (INT bit12)
           TBEN_L4_8IOL:O.Data[116].13   // IO-Link Port 8 - Output data word 2 (INT bit13)
           TBEN_L4_8IOL:O.Data[116].14   // IO-Link Port 8 - Output data word 2 (INT bit14)
           TBEN_L4_8IOL:O.Data[116].15   // IO-Link Port 8 - Output data word 2 (INT bit15)
           TBEN_L4_8IOL:O.Data[117]   // IO-Link Port 8 - Output data word 3
           TBEN_L4_8IOL:O.Data[117].0   // IO-Link Port 8 - Output data word 3 (INT bit0)
           TBEN_L4_8IOL:O.Data[117].1   // IO-Link Port 8 - Output data word 3 (INT bit1)
           TBEN_L4_8IOL:O.Data[117].2   // IO-Link Port 8 - Output data word 3 (INT bit2)
           TBEN_L4_8IOL:O.Data[117].3   // IO-Link Port 8 - Output data word 3 (INT bit3)
           TBEN_L4_8IOL:O.Data[117].4   // IO-Link Port 8 - Output data word 3 (INT bit4)
           TBEN_L4_8IOL:O.Data[117].5   // IO-Link Port 8 - Output data word 3 (INT bit5)
           TBEN_L4_8IOL:O.Data[117].6   // IO-Link Port 8 - Output data word 3 (INT bit6)
           TBEN_L4_8IOL:O.Data[117].7   // IO-Link Port 8 - Output data word 3 (INT bit7)
           TBEN_L4_8IOL:O.Data[117].8   // IO-Link Port 8 - Output data word 3 (INT bit8)
           TBEN_L4_8IOL:O.Data[117].9   // IO-Link Port 8 - Output data word 3 (INT bit9)
           TBEN_L4_8IOL:O.Data[117].10   // IO-Link Port 8 - Output data word 3 (INT bit10)
           TBEN_L4_8IOL:O.Data[117].11   // IO-Link Port 8 - Output data word 3 (INT bit11)
           TBEN_L4_8IOL:O.Data[117].12   // IO-Link Port 8 - Output data word 3 (INT bit12)
           TBEN_L4_8IOL:O.Data[117].13   // IO-Link Port 8 - Output data word 3 (INT bit13)
           TBEN_L4_8IOL:O.Data[117].14   // IO-Link Port 8 - Output data word 3 (INT bit14)
           TBEN_L4_8IOL:O.Data[117].15   // IO-Link Port 8 - Output data word 3 (INT bit15)
           TBEN_L4_8IOL:O.Data[118]   // IO-Link Port 8 - Output data word 4
           TBEN_L4_8IOL:O.Data[118].0   // IO-Link Port 8 - Output data word 4 (INT bit0)
           TBEN_L4_8IOL:O.Data[118].1   // IO-Link Port 8 - Output data word 4 (INT bit1)
           TBEN_L4_8IOL:O.Data[118].2   // IO-Link Port 8 - Output data word 4 (INT bit2)
           TBEN_L4_8IOL:O.Data[118].3   // IO-Link Port 8 - Output data word 4 (INT bit3)
           TBEN_L4_8IOL:O.Data[118].4   // IO-Link Port 8 - Output data word 4 (INT bit4)
           TBEN_L4_8IOL:O.Data[118].5   // IO-Link Port 8 - Output data word 4 (INT bit5)
           TBEN_L4_8IOL:O.Data[118].6   // IO-Link Port 8 - Output data word 4 (INT bit6)
           TBEN_L4_8IOL:O.Data[118].7   // IO-Link Port 8 - Output data word 4 (INT bit7)
           TBEN_L4_8IOL:O.Data[118].8   // IO-Link Port 8 - Output data word 4 (INT bit8)
           TBEN_L4_8IOL:O.Data[118].9   // IO-Link Port 8 - Output data word 4 (INT bit9)
           TBEN_L4_8IOL:O.Data[118].10   // IO-Link Port 8 - Output data word 4 (INT bit10)
           TBEN_L4_8IOL:O.Data[118].11   // IO-Link Port 8 - Output data word 4 (INT bit11)
           TBEN_L4_8IOL:O.Data[118].12   // IO-Link Port 8 - Output data word 4 (INT bit12)
           TBEN_L4_8IOL:O.Data[118].13   // IO-Link Port 8 - Output data word 4 (INT bit13)
           TBEN_L4_8IOL:O.Data[118].14   // IO-Link Port 8 - Output data word 4 (INT bit14)
           TBEN_L4_8IOL:O.Data[118].15   // IO-Link Port 8 - Output data word 4 (INT bit15)
           TBEN_L4_8IOL:O.Data[119]   // IO-Link Port 8 - Output data word 5
           TBEN_L4_8IOL:O.Data[119].0   // IO-Link Port 8 - Output data word 5 (INT bit0)
           TBEN_L4_8IOL:O.Data[119].1   // IO-Link Port 8 - Output data word 5 (INT bit1)
           TBEN_L4_8IOL:O.Data[119].2   // IO-Link Port 8 - Output data word 5 (INT bit2)
           TBEN_L4_8IOL:O.Data[119].3   // IO-Link Port 8 - Output data word 5 (INT bit3)
           TBEN_L4_8IOL:O.Data[119].4   // IO-Link Port 8 - Output data word 5 (INT bit4)
           TBEN_L4_8IOL:O.Data[119].5   // IO-Link Port 8 - Output data word 5 (INT bit5)
           TBEN_L4_8IOL:O.Data[119].6   // IO-Link Port 8 - Output data word 5 (INT bit6)
           TBEN_L4_8IOL:O.Data[119].7   // IO-Link Port 8 - Output data word 5 (INT bit7)
           TBEN_L4_8IOL:O.Data[119].8   // IO-Link Port 8 - Output data word 5 (INT bit8)
           TBEN_L4_8IOL:O.Data[119].9   // IO-Link Port 8 - Output data word 5 (INT bit9)
           TBEN_L4_8IOL:O.Data[119].10   // IO-Link Port 8 - Output data word 5 (INT bit10)
           TBEN_L4_8IOL:O.Data[119].11   // IO-Link Port 8 - Output data word 5 (INT bit11)
           TBEN_L4_8IOL:O.Data[119].12   // IO-Link Port 8 - Output data word 5 (INT bit12)
           TBEN_L4_8IOL:O.Data[119].13   // IO-Link Port 8 - Output data word 5 (INT bit13)
           TBEN_L4_8IOL:O.Data[119].14   // IO-Link Port 8 - Output data word 5 (INT bit14)
           TBEN_L4_8IOL:O.Data[119].15   // IO-Link Port 8 - Output data word 5 (INT bit15)
           TBEN_L4_8IOL:O.Data[120]   // IO-Link Port 8 - Output data word 6
           TBEN_L4_8IOL:O.Data[120].0   // IO-Link Port 8 - Output data word 6 (INT bit0)
           TBEN_L4_8IOL:O.Data[120].1   // IO-Link Port 8 - Output data word 6 (INT bit1)
           TBEN_L4_8IOL:O.Data[120].2   // IO-Link Port 8 - Output data word 6 (INT bit2)
           TBEN_L4_8IOL:O.Data[120].3   // IO-Link Port 8 - Output data word 6 (INT bit3)
           TBEN_L4_8IOL:O.Data[120].4   // IO-Link Port 8 - Output data word 6 (INT bit4)
           TBEN_L4_8IOL:O.Data[120].5   // IO-Link Port 8 - Output data word 6 (INT bit5)
           TBEN_L4_8IOL:O.Data[120].6   // IO-Link Port 8 - Output data word 6 (INT bit6)
           TBEN_L4_8IOL:O.Data[120].7   // IO-Link Port 8 - Output data word 6 (INT bit7)
           TBEN_L4_8IOL:O.Data[120].8   // IO-Link Port 8 - Output data word 6 (INT bit8)
           TBEN_L4_8IOL:O.Data[120].9   // IO-Link Port 8 - Output data word 6 (INT bit9)
           TBEN_L4_8IOL:O.Data[120].10   // IO-Link Port 8 - Output data word 6 (INT bit10)
           TBEN_L4_8IOL:O.Data[120].11   // IO-Link Port 8 - Output data word 6 (INT bit11)
           TBEN_L4_8IOL:O.Data[120].12   // IO-Link Port 8 - Output data word 6 (INT bit12)
           TBEN_L4_8IOL:O.Data[120].13   // IO-Link Port 8 - Output data word 6 (INT bit13)
           TBEN_L4_8IOL:O.Data[120].14   // IO-Link Port 8 - Output data word 6 (INT bit14)
           TBEN_L4_8IOL:O.Data[120].15   // IO-Link Port 8 - Output data word 6 (INT bit15)
           TBEN_L4_8IOL:O.Data[121]   // IO-Link Port 8 - Output data word 7
           TBEN_L4_8IOL:O.Data[121].0   // IO-Link Port 8 - Output data word 7 (INT bit0)
           TBEN_L4_8IOL:O.Data[121].1   // IO-Link Port 8 - Output data word 7 (INT bit1)
           TBEN_L4_8IOL:O.Data[121].2   // IO-Link Port 8 - Output data word 7 (INT bit2)
           TBEN_L4_8IOL:O.Data[121].3   // IO-Link Port 8 - Output data word 7 (INT bit3)
           TBEN_L4_8IOL:O.Data[121].4   // IO-Link Port 8 - Output data word 7 (INT bit4)
           TBEN_L4_8IOL:O.Data[121].5   // IO-Link Port 8 - Output data word 7 (INT bit5)
           TBEN_L4_8IOL:O.Data[121].6   // IO-Link Port 8 - Output data word 7 (INT bit6)
           TBEN_L4_8IOL:O.Data[121].7   // IO-Link Port 8 - Output data word 7 (INT bit7)
           TBEN_L4_8IOL:O.Data[121].8   // IO-Link Port 8 - Output data word 7 (INT bit8)
           TBEN_L4_8IOL:O.Data[121].9   // IO-Link Port 8 - Output data word 7 (INT bit9)
           TBEN_L4_8IOL:O.Data[121].10   // IO-Link Port 8 - Output data word 7 (INT bit10)
           TBEN_L4_8IOL:O.Data[121].11   // IO-Link Port 8 - Output data word 7 (INT bit11)
           TBEN_L4_8IOL:O.Data[121].12   // IO-Link Port 8 - Output data word 7 (INT bit12)
           TBEN_L4_8IOL:O.Data[121].13   // IO-Link Port 8 - Output data word 7 (INT bit13)
           TBEN_L4_8IOL:O.Data[121].14   // IO-Link Port 8 - Output data word 7 (INT bit14)
           TBEN_L4_8IOL:O.Data[121].15   // IO-Link Port 8 - Output data word 7 (INT bit15)
           TBEN_L4_8IOL:O.Data[122]   // IO-Link Port 8 - Output data word 8
           TBEN_L4_8IOL:O.Data[122].0   // IO-Link Port 8 - Output data word 8 (INT bit0)
           TBEN_L4_8IOL:O.Data[122].1   // IO-Link Port 8 - Output data word 8 (INT bit1)
           TBEN_L4_8IOL:O.Data[122].2   // IO-Link Port 8 - Output data word 8 (INT bit2)
           TBEN_L4_8IOL:O.Data[122].3   // IO-Link Port 8 - Output data word 8 (INT bit3)
           TBEN_L4_8IOL:O.Data[122].4   // IO-Link Port 8 - Output data word 8 (INT bit4)
           TBEN_L4_8IOL:O.Data[122].5   // IO-Link Port 8 - Output data word 8 (INT bit5)
           TBEN_L4_8IOL:O.Data[122].6   // IO-Link Port 8 - Output data word 8 (INT bit6)
           TBEN_L4_8IOL:O.Data[122].7   // IO-Link Port 8 - Output data word 8 (INT bit7)
           TBEN_L4_8IOL:O.Data[122].8   // IO-Link Port 8 - Output data word 8 (INT bit8)
           TBEN_L4_8IOL:O.Data[122].9   // IO-Link Port 8 - Output data word 8 (INT bit9)
           TBEN_L4_8IOL:O.Data[122].10   // IO-Link Port 8 - Output data word 8 (INT bit10)
           TBEN_L4_8IOL:O.Data[122].11   // IO-Link Port 8 - Output data word 8 (INT bit11)
           TBEN_L4_8IOL:O.Data[122].12   // IO-Link Port 8 - Output data word 8 (INT bit12)
           TBEN_L4_8IOL:O.Data[122].13   // IO-Link Port 8 - Output data word 8 (INT bit13)
           TBEN_L4_8IOL:O.Data[122].14   // IO-Link Port 8 - Output data word 8 (INT bit14)
           TBEN_L4_8IOL:O.Data[122].15   // IO-Link Port 8 - Output data word 8 (INT bit15)
           TBEN_L4_8IOL:O.Data[123]   // IO-Link Port 8 - Output data word 9
           TBEN_L4_8IOL:O.Data[123].0   // IO-Link Port 8 - Output data word 9 (INT bit0)
           TBEN_L4_8IOL:O.Data[123].1   // IO-Link Port 8 - Output data word 9 (INT bit1)
           TBEN_L4_8IOL:O.Data[123].2   // IO-Link Port 8 - Output data word 9 (INT bit2)
           TBEN_L4_8IOL:O.Data[123].3   // IO-Link Port 8 - Output data word 9 (INT bit3)
           TBEN_L4_8IOL:O.Data[123].4   // IO-Link Port 8 - Output data word 9 (INT bit4)
           TBEN_L4_8IOL:O.Data[123].5   // IO-Link Port 8 - Output data word 9 (INT bit5)
           TBEN_L4_8IOL:O.Data[123].6   // IO-Link Port 8 - Output data word 9 (INT bit6)
           TBEN_L4_8IOL:O.Data[123].7   // IO-Link Port 8 - Output data word 9 (INT bit7)
           TBEN_L4_8IOL:O.Data[123].8   // IO-Link Port 8 - Output data word 9 (INT bit8)
           TBEN_L4_8IOL:O.Data[123].9   // IO-Link Port 8 - Output data word 9 (INT bit9)
           TBEN_L4_8IOL:O.Data[123].10   // IO-Link Port 8 - Output data word 9 (INT bit10)
           TBEN_L4_8IOL:O.Data[123].11   // IO-Link Port 8 - Output data word 9 (INT bit11)
           TBEN_L4_8IOL:O.Data[123].12   // IO-Link Port 8 - Output data word 9 (INT bit12)
           TBEN_L4_8IOL:O.Data[123].13   // IO-Link Port 8 - Output data word 9 (INT bit13)
           TBEN_L4_8IOL:O.Data[123].14   // IO-Link Port 8 - Output data word 9 (INT bit14)
           TBEN_L4_8IOL:O.Data[123].15   // IO-Link Port 8 - Output data word 9 (INT bit15)
           TBEN_L4_8IOL:O.Data[124]   // IO-Link Port 8 - Output data word 10
           TBEN_L4_8IOL:O.Data[124].0   // IO-Link Port 8 - Output data word 10 (INT bit0)
           TBEN_L4_8IOL:O.Data[124].1   // IO-Link Port 8 - Output data word 10 (INT bit1)
           TBEN_L4_8IOL:O.Data[124].2   // IO-Link Port 8 - Output data word 10 (INT bit2)
           TBEN_L4_8IOL:O.Data[124].3   // IO-Link Port 8 - Output data word 10 (INT bit3)
           TBEN_L4_8IOL:O.Data[124].4   // IO-Link Port 8 - Output data word 10 (INT bit4)
           TBEN_L4_8IOL:O.Data[124].5   // IO-Link Port 8 - Output data word 10 (INT bit5)
           TBEN_L4_8IOL:O.Data[124].6   // IO-Link Port 8 - Output data word 10 (INT bit6)
           TBEN_L4_8IOL:O.Data[124].7   // IO-Link Port 8 - Output data word 10 (INT bit7)
           TBEN_L4_8IOL:O.Data[124].8   // IO-Link Port 8 - Output data word 10 (INT bit8)
           TBEN_L4_8IOL:O.Data[124].9   // IO-Link Port 8 - Output data word 10 (INT bit9)
           TBEN_L4_8IOL:O.Data[124].10   // IO-Link Port 8 - Output data word 10 (INT bit10)
           TBEN_L4_8IOL:O.Data[124].11   // IO-Link Port 8 - Output data word 10 (INT bit11)
           TBEN_L4_8IOL:O.Data[124].12   // IO-Link Port 8 - Output data word 10 (INT bit12)
           TBEN_L4_8IOL:O.Data[124].13   // IO-Link Port 8 - Output data word 10 (INT bit13)
           TBEN_L4_8IOL:O.Data[124].14   // IO-Link Port 8 - Output data word 10 (INT bit14)
           TBEN_L4_8IOL:O.Data[124].15   // IO-Link Port 8 - Output data word 10 (INT bit15)
           TBEN_L4_8IOL:O.Data[125]   // IO-Link Port 8 - Output data word 11
           TBEN_L4_8IOL:O.Data[125].0   // IO-Link Port 8 - Output data word 11 (INT bit0)
           TBEN_L4_8IOL:O.Data[125].1   // IO-Link Port 8 - Output data word 11 (INT bit1)
           TBEN_L4_8IOL:O.Data[125].2   // IO-Link Port 8 - Output data word 11 (INT bit2)
           TBEN_L4_8IOL:O.Data[125].3   // IO-Link Port 8 - Output data word 11 (INT bit3)
           TBEN_L4_8IOL:O.Data[125].4   // IO-Link Port 8 - Output data word 11 (INT bit4)
           TBEN_L4_8IOL:O.Data[125].5   // IO-Link Port 8 - Output data word 11 (INT bit5)
           TBEN_L4_8IOL:O.Data[125].6   // IO-Link Port 8 - Output data word 11 (INT bit6)
           TBEN_L4_8IOL:O.Data[125].7   // IO-Link Port 8 - Output data word 11 (INT bit7)
           TBEN_L4_8IOL:O.Data[125].8   // IO-Link Port 8 - Output data word 11 (INT bit8)
           TBEN_L4_8IOL:O.Data[125].9   // IO-Link Port 8 - Output data word 11 (INT bit9)
           TBEN_L4_8IOL:O.Data[125].10   // IO-Link Port 8 - Output data word 11 (INT bit10)
           TBEN_L4_8IOL:O.Data[125].11   // IO-Link Port 8 - Output data word 11 (INT bit11)
           TBEN_L4_8IOL:O.Data[125].12   // IO-Link Port 8 - Output data word 11 (INT bit12)
           TBEN_L4_8IOL:O.Data[125].13   // IO-Link Port 8 - Output data word 11 (INT bit13)
           TBEN_L4_8IOL:O.Data[125].14   // IO-Link Port 8 - Output data word 11 (INT bit14)
           TBEN_L4_8IOL:O.Data[125].15   // IO-Link Port 8 - Output data word 11 (INT bit15)
           TBEN_L4_8IOL:O.Data[126]   // IO-Link Port 8 - Output data word 12
           TBEN_L4_8IOL:O.Data[126].0   // IO-Link Port 8 - Output data word 12 (INT bit0)
           TBEN_L4_8IOL:O.Data[126].1   // IO-Link Port 8 - Output data word 12 (INT bit1)
           TBEN_L4_8IOL:O.Data[126].2   // IO-Link Port 8 - Output data word 12 (INT bit2)
           TBEN_L4_8IOL:O.Data[126].3   // IO-Link Port 8 - Output data word 12 (INT bit3)
           TBEN_L4_8IOL:O.Data[126].4   // IO-Link Port 8 - Output data word 12 (INT bit4)
           TBEN_L4_8IOL:O.Data[126].5   // IO-Link Port 8 - Output data word 12 (INT bit5)
           TBEN_L4_8IOL:O.Data[126].6   // IO-Link Port 8 - Output data word 12 (INT bit6)
           TBEN_L4_8IOL:O.Data[126].7   // IO-Link Port 8 - Output data word 12 (INT bit7)
           TBEN_L4_8IOL:O.Data[126].8   // IO-Link Port 8 - Output data word 12 (INT bit8)
           TBEN_L4_8IOL:O.Data[126].9   // IO-Link Port 8 - Output data word 12 (INT bit9)
           TBEN_L4_8IOL:O.Data[126].10   // IO-Link Port 8 - Output data word 12 (INT bit10)
           TBEN_L4_8IOL:O.Data[126].11   // IO-Link Port 8 - Output data word 12 (INT bit11)
           TBEN_L4_8IOL:O.Data[126].12   // IO-Link Port 8 - Output data word 12 (INT bit12)
           TBEN_L4_8IOL:O.Data[126].13   // IO-Link Port 8 - Output data word 12 (INT bit13)
           TBEN_L4_8IOL:O.Data[126].14   // IO-Link Port 8 - Output data word 12 (INT bit14)
           TBEN_L4_8IOL:O.Data[126].15   // IO-Link Port 8 - Output data word 12 (INT bit15)
           TBEN_L4_8IOL:O.Data[127]   // IO-Link Port 8 - Output data word 13
           TBEN_L4_8IOL:O.Data[127].0   // IO-Link Port 8 - Output data word 13 (INT bit0)
           TBEN_L4_8IOL:O.Data[127].1   // IO-Link Port 8 - Output data word 13 (INT bit1)
           TBEN_L4_8IOL:O.Data[127].2   // IO-Link Port 8 - Output data word 13 (INT bit2)
           TBEN_L4_8IOL:O.Data[127].3   // IO-Link Port 8 - Output data word 13 (INT bit3)
           TBEN_L4_8IOL:O.Data[127].4   // IO-Link Port 8 - Output data word 13 (INT bit4)
           TBEN_L4_8IOL:O.Data[127].5   // IO-Link Port 8 - Output data word 13 (INT bit5)
           TBEN_L4_8IOL:O.Data[127].6   // IO-Link Port 8 - Output data word 13 (INT bit6)
           TBEN_L4_8IOL:O.Data[127].7   // IO-Link Port 8 - Output data word 13 (INT bit7)
           TBEN_L4_8IOL:O.Data[127].8   // IO-Link Port 8 - Output data word 13 (INT bit8)
           TBEN_L4_8IOL:O.Data[127].9   // IO-Link Port 8 - Output data word 13 (INT bit9)
           TBEN_L4_8IOL:O.Data[127].10   // IO-Link Port 8 - Output data word 13 (INT bit10)
           TBEN_L4_8IOL:O.Data[127].11   // IO-Link Port 8 - Output data word 13 (INT bit11)
           TBEN_L4_8IOL:O.Data[127].12   // IO-Link Port 8 - Output data word 13 (INT bit12)
           TBEN_L4_8IOL:O.Data[127].13   // IO-Link Port 8 - Output data word 13 (INT bit13)
           TBEN_L4_8IOL:O.Data[127].14   // IO-Link Port 8 - Output data word 13 (INT bit14)
           TBEN_L4_8IOL:O.Data[127].15   // IO-Link Port 8 - Output data word 13 (INT bit15)
           TBEN_L4_8IOL:O.Data[128]   // IO-Link Port 8 - Output data word 14
           TBEN_L4_8IOL:O.Data[128].0   // IO-Link Port 8 - Output data word 14 (INT bit0)
           TBEN_L4_8IOL:O.Data[128].1   // IO-Link Port 8 - Output data word 14 (INT bit1)
           TBEN_L4_8IOL:O.Data[128].2   // IO-Link Port 8 - Output data word 14 (INT bit2)
           TBEN_L4_8IOL:O.Data[128].3   // IO-Link Port 8 - Output data word 14 (INT bit3)
           TBEN_L4_8IOL:O.Data[128].4   // IO-Link Port 8 - Output data word 14 (INT bit4)
           TBEN_L4_8IOL:O.Data[128].5   // IO-Link Port 8 - Output data word 14 (INT bit5)
           TBEN_L4_8IOL:O.Data[128].6   // IO-Link Port 8 - Output data word 14 (INT bit6)
           TBEN_L4_8IOL:O.Data[128].7   // IO-Link Port 8 - Output data word 14 (INT bit7)
           TBEN_L4_8IOL:O.Data[128].8   // IO-Link Port 8 - Output data word 14 (INT bit8)
           TBEN_L4_8IOL:O.Data[128].9   // IO-Link Port 8 - Output data word 14 (INT bit9)
           TBEN_L4_8IOL:O.Data[128].10   // IO-Link Port 8 - Output data word 14 (INT bit10)
           TBEN_L4_8IOL:O.Data[128].11   // IO-Link Port 8 - Output data word 14 (INT bit11)
           TBEN_L4_8IOL:O.Data[128].12   // IO-Link Port 8 - Output data word 14 (INT bit12)
           TBEN_L4_8IOL:O.Data[128].13   // IO-Link Port 8 - Output data word 14 (INT bit13)
           TBEN_L4_8IOL:O.Data[128].14   // IO-Link Port 8 - Output data word 14 (INT bit14)
           TBEN_L4_8IOL:O.Data[128].15   // IO-Link Port 8 - Output data word 14 (INT bit15)
           TBEN_L4_8IOL:O.Data[129]   // IO-Link Port 8 - Output data word 15
           TBEN_L4_8IOL:O.Data[129].0   // IO-Link Port 8 - Output data word 15 (INT bit0)
           TBEN_L4_8IOL:O.Data[129].1   // IO-Link Port 8 - Output data word 15 (INT bit1)
           TBEN_L4_8IOL:O.Data[129].2   // IO-Link Port 8 - Output data word 15 (INT bit2)
           TBEN_L4_8IOL:O.Data[129].3   // IO-Link Port 8 - Output data word 15 (INT bit3)
           TBEN_L4_8IOL:O.Data[129].4   // IO-Link Port 8 - Output data word 15 (INT bit4)
           TBEN_L4_8IOL:O.Data[129].5   // IO-Link Port 8 - Output data word 15 (INT bit5)
           TBEN_L4_8IOL:O.Data[129].6   // IO-Link Port 8 - Output data word 15 (INT bit6)
           TBEN_L4_8IOL:O.Data[129].7   // IO-Link Port 8 - Output data word 15 (INT bit7)
           TBEN_L4_8IOL:O.Data[129].8   // IO-Link Port 8 - Output data word 15 (INT bit8)
           TBEN_L4_8IOL:O.Data[129].9   // IO-Link Port 8 - Output data word 15 (INT bit9)
           TBEN_L4_8IOL:O.Data[129].10   // IO-Link Port 8 - Output data word 15 (INT bit10)
           TBEN_L4_8IOL:O.Data[129].11   // IO-Link Port 8 - Output data word 15 (INT bit11)
           TBEN_L4_8IOL:O.Data[129].12   // IO-Link Port 8 - Output data word 15 (INT bit12)
           TBEN_L4_8IOL:O.Data[129].13   // IO-Link Port 8 - Output data word 15 (INT bit13)
           TBEN_L4_8IOL:O.Data[129].14   // IO-Link Port 8 - Output data word 15 (INT bit14)
           TBEN_L4_8IOL:O.Data[129].15   // IO-Link Port 8 - Output data word 15 (INT bit15)
           TBEN_L4_8IOL:O.Data[130]   // VAUX1 Pin1 C0 (Ch0/1), VAUX1 Pin1 C1 (Ch2/3), VAUX1 Pin1 C2 (Ch4/5), VAUX1 Pin1 C3 (Ch6/7), VAUX1 Pin1 C4 (Ch8), VAUX1 Pin1 C5 (Ch10), VAUX1 Pin1 C6 (Ch12), VAUX1 Pin1 C7 (Ch14), VAUX2 Pin2 C4 (Ch9), VAUX2 Pin2 C5 (Ch11), VAUX2 Pin2 C6 (Ch13), VAUX2 Pin2 C7 (Ch15)
           TBEN_L4_8IOL:O.Data[130].0   // VAUX1 Pin1 C0 (Ch0/1) (ENUM bit0): 0=off, 1=on
           TBEN_L4_8IOL:O.Data[130].1   // VAUX1 Pin1 C1 (Ch2/3) (ENUM bit0): 0=off, 1=on
           TBEN_L4_8IOL:O.Data[130].2   // VAUX1 Pin1 C2 (Ch4/5) (ENUM bit0): 0=off, 1=on
           TBEN_L4_8IOL:O.Data[130].3   // VAUX1 Pin1 C3 (Ch6/7) (ENUM bit0): 0=off, 1=on
           TBEN_L4_8IOL:O.Data[130].4   // VAUX1 Pin1 C4 (Ch8) (ENUM bit0): 0=off, 1=on
           TBEN_L4_8IOL:O.Data[130].5   // VAUX1 Pin1 C5 (Ch10) (ENUM bit0): 0=off, 1=on
           TBEN_L4_8IOL:O.Data[130].6   // VAUX1 Pin1 C6 (Ch12) (ENUM bit0): 0=off, 1=on
           TBEN_L4_8IOL:O.Data[130].7   // VAUX1 Pin1 C7 (Ch14) (ENUM bit0): 0=off, 1=on
           TBEN_L4_8IOL:O.Data[130].8   // Reserved
           TBEN_L4_8IOL:O.Data[130].9   // Reserved
           TBEN_L4_8IOL:O.Data[130].10   // Reserved
           TBEN_L4_8IOL:O.Data[130].11   // Reserved
           TBEN_L4_8IOL:O.Data[130].12   // VAUX2 Pin2 C4 (Ch9) (ENUM bit0): 0=off, 1=on
           TBEN_L4_8IOL:O.Data[130].13   // VAUX2 Pin2 C5 (Ch11) (ENUM bit0): 0=off, 1=on
           TBEN_L4_8IOL:O.Data[130].14   // VAUX2 Pin2 C6 (Ch13) (ENUM bit0): 0=off, 1=on
           TBEN_L4_8IOL:O.Data[130].15   // VAUX2 Pin2 C7 (Ch15) (ENUM bit0): 0=off, 1=on
           TBEN_L4_8IOL:C.Data[0]   // Reserved
           TBEN_L4_8IOL:C.Data[1]   // Reserved
           TBEN_L4_8IOL:C.Data[2]   // Reserved
           TBEN_L4_8IOL:C.Data[3]   // Reserved
           TBEN_L4_8IOL:C.Data[4]   // Reserved
           TBEN_L4_8IOL:C.Data[5]   // Reserved
           TBEN_L4_8IOL:C.Data[6]   // Reserved
           TBEN_L4_8IOL:C.Data[7]   // Reserved
           TBEN_L4_8IOL:C.Data[8]   // Reserved
           TBEN_L4_8IOL:C.Data[9]   // Quick Connect, Eth Custom Setup, LED-behavior (PWR) at V2 undervoltage
           TBEN_L4_8IOL:C.Data[9].0   // Quick Connect: 0=disable, 1=enable
           TBEN_L4_8IOL:C.Data[9].1   // Eth 1 Custom Setup: 0=Auto-negotiate, 1=100BT/FD
           TBEN_L4_8IOL:C.Data[9].2   // Eth 2 Custom Setup: 0=Auto-negotiate, 1=100BT/FD
           TBEN_L4_8IOL:C.Data[9].3   // LED-behavior (PWR) at V2 undervoltage: 0=Red, 1=Green
           TBEN_L4_8IOL:C.Data[9].4   // Reserved
           TBEN_L4_8IOL:C.Data[9].5   // Reserved
           TBEN_L4_8IOL:C.Data[9].6   // Reserved
           TBEN_L4_8IOL:C.Data[9].7   // Reserved
           TBEN_L4_8IOL:C.Data[10]   // DXP 1 - Manual reset after overcurr.
           TBEN_L4_8IOL:C.Data[10].0   // DXP 1 - Manual reset after overcurr. (ENUM bit0): 0=no, 1=yes
           TBEN_L4_8IOL:C.Data[10].1   // Reserved
           TBEN_L4_8IOL:C.Data[10].2   // Reserved
           TBEN_L4_8IOL:C.Data[10].3   // Reserved
           TBEN_L4_8IOL:C.Data[10].4   // Reserved
           TBEN_L4_8IOL:C.Data[10].5   // Reserved
           TBEN_L4_8IOL:C.Data[10].6   // Reserved
           TBEN_L4_8IOL:C.Data[10].7   // Reserved
           TBEN_L4_8IOL:C.Data[11]   // DXP 3 - Manual reset after overcurr.
           TBEN_L4_8IOL:C.Data[11].0   // DXP 3 - Manual reset after overcurr. (ENUM bit0): 0=no, 1=yes
           TBEN_L4_8IOL:C.Data[11].1   // Reserved
           TBEN_L4_8IOL:C.Data[11].2   // Reserved
           TBEN_L4_8IOL:C.Data[11].3   // Reserved
           TBEN_L4_8IOL:C.Data[11].4   // Reserved
           TBEN_L4_8IOL:C.Data[11].5   // Reserved
           TBEN_L4_8IOL:C.Data[11].6   // Reserved
           TBEN_L4_8IOL:C.Data[11].7   // Reserved
           TBEN_L4_8IOL:C.Data[12]   // DXP 5 - Manual reset after overcurr.
           TBEN_L4_8IOL:C.Data[12].0   // DXP 5 - Manual reset after overcurr. (ENUM bit0): 0=no, 1=yes
           TBEN_L4_8IOL:C.Data[12].1   // Reserved
           TBEN_L4_8IOL:C.Data[12].2   // Reserved
           TBEN_L4_8IOL:C.Data[12].3   // Reserved
           TBEN_L4_8IOL:C.Data[12].4   // Reserved
           TBEN_L4_8IOL:C.Data[12].5   // Reserved
           TBEN_L4_8IOL:C.Data[12].6   // Reserved
           TBEN_L4_8IOL:C.Data[12].7   // Reserved
           TBEN_L4_8IOL:C.Data[13]   // DXP 7 - Manual reset after overcurr.
           TBEN_L4_8IOL:C.Data[13].0   // DXP 7 - Manual reset after overcurr. (ENUM bit0): 0=no, 1=yes
           TBEN_L4_8IOL:C.Data[13].1   // Reserved
           TBEN_L4_8IOL:C.Data[13].2   // Reserved
           TBEN_L4_8IOL:C.Data[13].3   // Reserved
           TBEN_L4_8IOL:C.Data[13].4   // Reserved
           TBEN_L4_8IOL:C.Data[13].5   // Reserved
           TBEN_L4_8IOL:C.Data[13].6   // Reserved
           TBEN_L4_8IOL:C.Data[13].7   // Reserved
           TBEN_L4_8IOL:C.Data[14]   // DXP 1 - Activate output
           TBEN_L4_8IOL:C.Data[14].0   // DXP 1 - Activate output (ENUM bit0): 0=no, 1=yes
           TBEN_L4_8IOL:C.Data[14].1   // Reserved
           TBEN_L4_8IOL:C.Data[14].2   // Reserved
           TBEN_L4_8IOL:C.Data[14].3   // Reserved
           TBEN_L4_8IOL:C.Data[14].4   // Reserved
           TBEN_L4_8IOL:C.Data[14].5   // Reserved
           TBEN_L4_8IOL:C.Data[14].6   // Reserved
           TBEN_L4_8IOL:C.Data[14].7   // Reserved
           TBEN_L4_8IOL:C.Data[15]   // DXP 3 - Activate output
           TBEN_L4_8IOL:C.Data[15].0   // DXP 3 - Activate output (ENUM bit0): 0=no, 1=yes
           TBEN_L4_8IOL:C.Data[15].1   // Reserved
           TBEN_L4_8IOL:C.Data[15].2   // Reserved
           TBEN_L4_8IOL:C.Data[15].3   // Reserved
           TBEN_L4_8IOL:C.Data[15].4   // Reserved
           TBEN_L4_8IOL:C.Data[15].5   // Reserved
           TBEN_L4_8IOL:C.Data[15].6   // Reserved
           TBEN_L4_8IOL:C.Data[15].7   // Reserved
           TBEN_L4_8IOL:C.Data[16]   // DXP 5 - Activate output
           TBEN_L4_8IOL:C.Data[16].0   // DXP 5 - Activate output (ENUM bit0): 0=no, 1=yes
           TBEN_L4_8IOL:C.Data[16].1   // Reserved
           TBEN_L4_8IOL:C.Data[16].2   // Reserved
           TBEN_L4_8IOL:C.Data[16].3   // Reserved
           TBEN_L4_8IOL:C.Data[16].4   // Reserved
           TBEN_L4_8IOL:C.Data[16].5   // Reserved
           TBEN_L4_8IOL:C.Data[16].6   // Reserved
           TBEN_L4_8IOL:C.Data[16].7   // Reserved
           TBEN_L4_8IOL:C.Data[17]   // DXP 7 - Activate output
           TBEN_L4_8IOL:C.Data[17].0   // DXP 7 - Activate output (ENUM bit0): 0=no, 1=yes
           TBEN_L4_8IOL:C.Data[17].1   // Reserved
           TBEN_L4_8IOL:C.Data[17].2   // Reserved
           TBEN_L4_8IOL:C.Data[17].3   // Reserved
           TBEN_L4_8IOL:C.Data[17].4   // Reserved
           TBEN_L4_8IOL:C.Data[17].5   // Reserved
           TBEN_L4_8IOL:C.Data[17].6   // Reserved
           TBEN_L4_8IOL:C.Data[17].7   // Reserved
           TBEN_L4_8IOL:C.Data[18]   // IO-Link Port 1 - Operation mode
           TBEN_L4_8IOL:C.Data[18].0   // IO-Link Port 1 - Operation mode (ENUM bit0): 0000=IO-Link without validation, 0001=IO-Link with family compatible device
           TBEN_L4_8IOL:C.Data[18].1   // IO-Link Port 1 - Operation mode (ENUM bit1): 0010=IO-Link with compatible device, 0011=IO-Link with identical device
           TBEN_L4_8IOL:C.Data[18].2   // IO-Link Port 1 - Operation mode (ENUM bit2): 0100=DI (with parameter access)
           TBEN_L4_8IOL:C.Data[18].3   // IO-Link Port 1 - Operation mode (ENUM bit3): 1000=DI
           TBEN_L4_8IOL:C.Data[18].4   // Reserved
           TBEN_L4_8IOL:C.Data[18].5   // Reserved
           TBEN_L4_8IOL:C.Data[18].6   // Reserved
           TBEN_L4_8IOL:C.Data[18].7   // Reserved
           TBEN_L4_8IOL:C.Data[19]   // IO-Link Port 1 - Data storage mode
           TBEN_L4_8IOL:C.Data[19].0   // IO-Link Port 1 - Data storage mode (ENUM bit0): 00=activated, 01=overwrite
           TBEN_L4_8IOL:C.Data[19].1   // IO-Link Port 1 - Data storage mode (ENUM bit1): 10=read in, 11=deactivated, clear
           TBEN_L4_8IOL:C.Data[19].2   // Reserved
           TBEN_L4_8IOL:C.Data[19].3   // Reserved
           TBEN_L4_8IOL:C.Data[19].4   // Reserved
           TBEN_L4_8IOL:C.Data[19].5   // Reserved
           TBEN_L4_8IOL:C.Data[19].6   // Reserved
           TBEN_L4_8IOL:C.Data[19].7   // Reserved
           TBEN_L4_8IOL:C.Data[20]   // IO-Link Port 1 - Cycle time
           TBEN_L4_8IOL:C.Data[20].0   // IO-Link Port 1 - Cycle time (ENUM bit0): 00000000=automatic, 00010000=1.6 ms, 00011000=2.4 ms, 00100000=3.2 ms, 00101000=4.0 ms, 00110000=4.8 ms, 00111000=5.6 ms, 01000000=6.4 ms, 01000010=7.2 ms, 01000100=8.0 ms, 01000110=8.8 ms, 01001000=9.6 ms
           TBEN_L4_8IOL:C.Data[20].1   // IO-Link Port 1 - Cycle time (ENUM bit1): 01001010=10.4 ms, 01001100=11.2 ms, 01001110=12.0 ms, 01010000=12.8 ms, 01010100=14.4 ms, 01011000=16.0 ms, 01011100=17.6 ms, 01100000=19.2 ms, 01100100=20.8 ms, 01101000=22.4 ms, 01101100=24.0 ms, 01110000=25.6 ms
           TBEN_L4_8IOL:C.Data[20].2   // IO-Link Port 1 - Cycle time (ENUM bit2): 01110100=27.2 ms, 01111000=28.8 ms, 01111100=30.4 ms, 10000000=32.0 ms, 10000001=33.6 ms, 10000010=35.2 ms, 10000011=36.8 ms, 10000100=38.4 ms, 10000101=40.0 ms, 10000110=41.6 ms, 10000111=43.2 ms, 10001000=44.8 ms
           TBEN_L4_8IOL:C.Data[20].3   // IO-Link Port 1 - Cycle time (ENUM bit3): 10001001=46.4 ms, 10001010=48.0 ms, 10001011=49.6 ms, 10001100=51.2 ms, 10001101=52.8 ms, 10001110=54.4 ms, 10001111=56.0 ms, 10010000=57.6 ms, 10010001=59.2 ms, 10010010=60.8 ms, 10010011=62.4 ms, 10010100=64.0 ms
           TBEN_L4_8IOL:C.Data[20].4   // IO-Link Port 1 - Cycle time (ENUM bit4): 10010101=65.6 ms, 10010110=67.2 ms, 10010111=68.8 ms, 10011000=70.4 ms, 10011001=72.0 ms, 10011010=73.6 ms, 10011011=75.2 ms, 10011100=76.8 ms, 10011101=78.4 ms, 10011110=80.0 ms, 10011111=81.6 ms
           TBEN_L4_8IOL:C.Data[20].5   // IO-Link Port 1 - Cycle time (ENUM bit5): 10100000=83.2 ms, 10100001=84.8 ms, 10100010=86.4 ms, 10100011=88.0 ms, 10100100=89.6 ms, 10100101=91.2 ms, 10100110=92.8 ms, 10100111=94.4 ms, 10101000=96.0 ms, 10101001=97.6 ms, 10101010=99.2 ms
           TBEN_L4_8IOL:C.Data[20].6   // IO-Link Port 1 - Cycle time (ENUM bit6): 10101011=100.8 ms, 10101100=102.4 ms, 10101101=104.0 ms, 10101110=105.6 ms, 10101111=107.2 ms, 10110000=108.8 ms, 10110001=110.4 ms, 10110010=112.0 ms, 10110011=113.6 ms, 10110100=115.2 ms, 10110101=116.8 ms
           TBEN_L4_8IOL:C.Data[20].7   // IO-Link Port 1 - Cycle time (ENUM bit7): 10110110=118.4 ms, 10110111=120.0 ms, 10111000=121.6 ms, 10111001=123.2 ms, 10111010=124.8 ms, 10111011=126.4 ms, 10111100=128.0 ms, 10111101=129.6 ms, 10111110=131.2 ms, 10111111=132.8 ms, 11111111=automatic, compatible
           TBEN_L4_8IOL:C.Data[21]   // IO-Link Port 1 - Revision
           TBEN_L4_8IOL:C.Data[21].0   // IO-Link Port 1 - Revision (ENUM bit0): 0=automatic, 1=V1.0
           TBEN_L4_8IOL:C.Data[21].1   // Reserved
           TBEN_L4_8IOL:C.Data[21].2   // Reserved
           TBEN_L4_8IOL:C.Data[21].3   // Reserved
           TBEN_L4_8IOL:C.Data[21].4   // Reserved
           TBEN_L4_8IOL:C.Data[21].5   // Reserved
           TBEN_L4_8IOL:C.Data[21].6   // Reserved
           TBEN_L4_8IOL:C.Data[21].7   // Reserved
           TBEN_L4_8IOL:C.Data[22]   // IO-Link Port 1 - Activate Quick Start-Up
           TBEN_L4_8IOL:C.Data[22].0   // IO-Link Port 1 - Activate Quick Start-Up (ENUM bit0): 0=no, 1=yes
           TBEN_L4_8IOL:C.Data[22].1   // Reserved
           TBEN_L4_8IOL:C.Data[22].2   // Reserved
           TBEN_L4_8IOL:C.Data[22].3   // Reserved
           TBEN_L4_8IOL:C.Data[22].4   // Reserved
           TBEN_L4_8IOL:C.Data[22].5   // Reserved
           TBEN_L4_8IOL:C.Data[22].6   // Reserved
           TBEN_L4_8IOL:C.Data[22].7   // Reserved
           TBEN_L4_8IOL:C.Data[23]   // IO-Link Port 1 - Device parametrization via GSD
           TBEN_L4_8IOL:C.Data[23].0   // IO-Link Port 1 - Device parametrization via GSD (ENUM bit0): 0=inactive, 1=active
           TBEN_L4_8IOL:C.Data[23].1   // Reserved
           TBEN_L4_8IOL:C.Data[23].2   // Reserved
           TBEN_L4_8IOL:C.Data[23].3   // Reserved
           TBEN_L4_8IOL:C.Data[23].4   // Reserved
           TBEN_L4_8IOL:C.Data[23].5   // Reserved
           TBEN_L4_8IOL:C.Data[23].6   // Reserved
           TBEN_L4_8IOL:C.Data[23].7   // Reserved
           TBEN_L4_8IOL:C.Data[24]   // IO-Link Port 1 - Process input data invalid
           TBEN_L4_8IOL:C.Data[24].0   // IO-Link Port 1 - Process input data invalid (ENUM bit0): 0=diagnostic generated, 1=no diagnostic generated
           TBEN_L4_8IOL:C.Data[24].1   // Reserved
           TBEN_L4_8IOL:C.Data[24].2   // Reserved
           TBEN_L4_8IOL:C.Data[24].3   // Reserved
           TBEN_L4_8IOL:C.Data[24].4   // Reserved
           TBEN_L4_8IOL:C.Data[24].5   // Reserved
           TBEN_L4_8IOL:C.Data[24].6   // Reserved
           TBEN_L4_8IOL:C.Data[24].7   // Reserved
           TBEN_L4_8IOL:C.Data[25]   // IO-Link Port 1 - Deactivate diagnostics
           TBEN_L4_8IOL:C.Data[25].0   // IO-Link Port 1 - Deactivate diagnostics (ENUM bit0): 00=no, 01=notifications
           TBEN_L4_8IOL:C.Data[25].1   // IO-Link Port 1 - Deactivate diagnostics (ENUM bit1): 10=notifications and warnings, 11=yes
           TBEN_L4_8IOL:C.Data[25].2   // Reserved
           TBEN_L4_8IOL:C.Data[25].3   // Reserved
           TBEN_L4_8IOL:C.Data[25].4   // Reserved
           TBEN_L4_8IOL:C.Data[25].5   // Reserved
           TBEN_L4_8IOL:C.Data[25].6   // Reserved
           TBEN_L4_8IOL:C.Data[25].7   // Reserved
           TBEN_L4_8IOL:C.Data[26]   // IO-Link Port 1 - Input data mapping
           TBEN_L4_8IOL:C.Data[26].0   // IO-Link Port 1 - Input data mapping (ENUM bit0): 00=direct, 01=swap 16 bit
           TBEN_L4_8IOL:C.Data[26].1   // IO-Link Port 1 - Input data mapping (ENUM bit1): 10=swap 32 bit, 11=swap
           TBEN_L4_8IOL:C.Data[26].2   // Reserved
           TBEN_L4_8IOL:C.Data[26].3   // Reserved
           TBEN_L4_8IOL:C.Data[26].4   // Reserved
           TBEN_L4_8IOL:C.Data[26].5   // Reserved
           TBEN_L4_8IOL:C.Data[26].6   // Reserved
           TBEN_L4_8IOL:C.Data[26].7   // Reserved
           TBEN_L4_8IOL:C.Data[27]   // IO-Link Port 1 - Output data mapping
           TBEN_L4_8IOL:C.Data[27].0   // IO-Link Port 1 - Output data mapping (ENUM bit0): 00=direct, 01=swap 16 bit
           TBEN_L4_8IOL:C.Data[27].1   // IO-Link Port 1 - Output data mapping (ENUM bit1): 10=swap 32 bit, 11=swap
           TBEN_L4_8IOL:C.Data[27].2   // Reserved
           TBEN_L4_8IOL:C.Data[27].3   // Reserved
           TBEN_L4_8IOL:C.Data[27].4   // Reserved
           TBEN_L4_8IOL:C.Data[27].5   // Reserved
           TBEN_L4_8IOL:C.Data[27].6   // Reserved
           TBEN_L4_8IOL:C.Data[27].7   // Reserved
           TBEN_L4_8IOL:C.Data[28]   // IO-Link Port 1 - Vendor ID
           TBEN_L4_8IOL:C.Data[28].0   // IO-Link Port 1 - Vendor ID (INT bit0)
           TBEN_L4_8IOL:C.Data[28].1   // IO-Link Port 1 - Vendor ID (INT bit1)
           TBEN_L4_8IOL:C.Data[28].2   // IO-Link Port 1 - Vendor ID (INT bit2)
           TBEN_L4_8IOL:C.Data[28].3   // IO-Link Port 1 - Vendor ID (INT bit3)
           TBEN_L4_8IOL:C.Data[28].4   // IO-Link Port 1 - Vendor ID (INT bit4)
           TBEN_L4_8IOL:C.Data[28].5   // IO-Link Port 1 - Vendor ID (INT bit5)
           TBEN_L4_8IOL:C.Data[28].6   // IO-Link Port 1 - Vendor ID (INT bit6)
           TBEN_L4_8IOL:C.Data[28].7   // IO-Link Port 1 - Vendor ID (INT bit7)
           TBEN_L4_8IOL:C.Data[29]   // IO-Link Port 1 - Vendor ID
           TBEN_L4_8IOL:C.Data[29].0   // IO-Link Port 1 - Vendor ID (INT bit8)
           TBEN_L4_8IOL:C.Data[29].1   // IO-Link Port 1 - Vendor ID (INT bit9)
           TBEN_L4_8IOL:C.Data[29].2   // IO-Link Port 1 - Vendor ID (INT bit10)
           TBEN_L4_8IOL:C.Data[29].3   // IO-Link Port 1 - Vendor ID (INT bit11)
           TBEN_L4_8IOL:C.Data[29].4   // IO-Link Port 1 - Vendor ID (INT bit12)
           TBEN_L4_8IOL:C.Data[29].5   // IO-Link Port 1 - Vendor ID (INT bit13)
           TBEN_L4_8IOL:C.Data[29].6   // IO-Link Port 1 - Vendor ID (INT bit14)
           TBEN_L4_8IOL:C.Data[29].7   // IO-Link Port 1 - Vendor ID (INT bit15)
           TBEN_L4_8IOL:C.Data[30]   // IO-Link Port 1 - Device ID
           TBEN_L4_8IOL:C.Data[30].0   // IO-Link Port 1 - Device ID (INT bit0)
           TBEN_L4_8IOL:C.Data[30].1   // IO-Link Port 1 - Device ID (INT bit1)
           TBEN_L4_8IOL:C.Data[30].2   // IO-Link Port 1 - Device ID (INT bit2)
           TBEN_L4_8IOL:C.Data[30].3   // IO-Link Port 1 - Device ID (INT bit3)
           TBEN_L4_8IOL:C.Data[30].4   // IO-Link Port 1 - Device ID (INT bit4)
           TBEN_L4_8IOL:C.Data[30].5   // IO-Link Port 1 - Device ID (INT bit5)
           TBEN_L4_8IOL:C.Data[30].6   // IO-Link Port 1 - Device ID (INT bit6)
           TBEN_L4_8IOL:C.Data[30].7   // IO-Link Port 1 - Device ID (INT bit7)
           TBEN_L4_8IOL:C.Data[31]   // IO-Link Port 1 - Device ID
           TBEN_L4_8IOL:C.Data[31].0   // IO-Link Port 1 - Device ID (INT bit8)
           TBEN_L4_8IOL:C.Data[31].1   // IO-Link Port 1 - Device ID (INT bit9)
           TBEN_L4_8IOL:C.Data[31].2   // IO-Link Port 1 - Device ID (INT bit10)
           TBEN_L4_8IOL:C.Data[31].3   // IO-Link Port 1 - Device ID (INT bit11)
           TBEN_L4_8IOL:C.Data[31].4   // IO-Link Port 1 - Device ID (INT bit12)
           TBEN_L4_8IOL:C.Data[31].5   // IO-Link Port 1 - Device ID (INT bit13)
           TBEN_L4_8IOL:C.Data[31].6   // IO-Link Port 1 - Device ID (INT bit14)
           TBEN_L4_8IOL:C.Data[31].7   // IO-Link Port 1 - Device ID (INT bit15)
           TBEN_L4_8IOL:C.Data[32]   // IO-Link Port 1 - Device ID
           TBEN_L4_8IOL:C.Data[32].0   // IO-Link Port 1 - Device ID (INT bit16)
           TBEN_L4_8IOL:C.Data[32].1   // IO-Link Port 1 - Device ID (INT bit17)
           TBEN_L4_8IOL:C.Data[32].2   // IO-Link Port 1 - Device ID (INT bit18)
           TBEN_L4_8IOL:C.Data[32].3   // IO-Link Port 1 - Device ID (INT bit19)
           TBEN_L4_8IOL:C.Data[32].4   // IO-Link Port 1 - Device ID (INT bit20)
           TBEN_L4_8IOL:C.Data[32].5   // IO-Link Port 1 - Device ID (INT bit21)
           TBEN_L4_8IOL:C.Data[32].6   // IO-Link Port 1 - Device ID (INT bit22)
           TBEN_L4_8IOL:C.Data[32].7   // IO-Link Port 1 - Device ID (INT bit23)
           TBEN_L4_8IOL:C.Data[33]   // IO-Link Port 1 - Device ID
           TBEN_L4_8IOL:C.Data[33].0   // IO-Link Port 1 - Device ID (INT bit24)
           TBEN_L4_8IOL:C.Data[33].1   // IO-Link Port 1 - Device ID (INT bit25)
           TBEN_L4_8IOL:C.Data[33].2   // IO-Link Port 1 - Device ID (INT bit26)
           TBEN_L4_8IOL:C.Data[33].3   // IO-Link Port 1 - Device ID (INT bit27)
           TBEN_L4_8IOL:C.Data[33].4   // IO-Link Port 1 - Device ID (INT bit28)
           TBEN_L4_8IOL:C.Data[33].5   // IO-Link Port 1 - Device ID (INT bit29)
           TBEN_L4_8IOL:C.Data[33].6   // IO-Link Port 1 - Device ID (INT bit30)
           TBEN_L4_8IOL:C.Data[33].7   // IO-Link Port 1 - Device ID (INT bit31)
           TBEN_L4_8IOL:C.Data[34]   // IO-Link Port 2 - Operation mode
           TBEN_L4_8IOL:C.Data[34].0   // IO-Link Port 2 - Operation mode (ENUM bit0): 0000=IO-Link without validation, 0001=IO-Link with family compatible device
           TBEN_L4_8IOL:C.Data[34].1   // IO-Link Port 2 - Operation mode (ENUM bit1): 0010=IO-Link with compatible device, 0011=IO-Link with identical device
           TBEN_L4_8IOL:C.Data[34].2   // IO-Link Port 2 - Operation mode (ENUM bit2): 0100=DI (with parameter access)
           TBEN_L4_8IOL:C.Data[34].3   // IO-Link Port 2 - Operation mode (ENUM bit3): 1000=DI
           TBEN_L4_8IOL:C.Data[34].4   // Reserved
           TBEN_L4_8IOL:C.Data[34].5   // Reserved
           TBEN_L4_8IOL:C.Data[34].6   // Reserved
           TBEN_L4_8IOL:C.Data[34].7   // Reserved
           TBEN_L4_8IOL:C.Data[35]   // IO-Link Port 2 - Data storage mode
           TBEN_L4_8IOL:C.Data[35].0   // IO-Link Port 2 - Data storage mode (ENUM bit0): 00=activated, 01=overwrite
           TBEN_L4_8IOL:C.Data[35].1   // IO-Link Port 2 - Data storage mode (ENUM bit1): 10=read in, 11=deactivated, clear
           TBEN_L4_8IOL:C.Data[35].2   // Reserved
           TBEN_L4_8IOL:C.Data[35].3   // Reserved
           TBEN_L4_8IOL:C.Data[35].4   // Reserved
           TBEN_L4_8IOL:C.Data[35].5   // Reserved
           TBEN_L4_8IOL:C.Data[35].6   // Reserved
           TBEN_L4_8IOL:C.Data[35].7   // Reserved
           TBEN_L4_8IOL:C.Data[36]   // IO-Link Port 2 - Cycle time
           TBEN_L4_8IOL:C.Data[36].0   // IO-Link Port 2 - Cycle time (ENUM bit0): 00000000=automatic, 00010000=1.6 ms, 00011000=2.4 ms, 00100000=3.2 ms, 00101000=4.0 ms, 00110000=4.8 ms, 00111000=5.6 ms, 01000000=6.4 ms, 01000010=7.2 ms, 01000100=8.0 ms, 01000110=8.8 ms, 01001000=9.6 ms
           TBEN_L4_8IOL:C.Data[36].1   // IO-Link Port 2 - Cycle time (ENUM bit1): 01001010=10.4 ms, 01001100=11.2 ms, 01001110=12.0 ms, 01010000=12.8 ms, 01010100=14.4 ms, 01011000=16.0 ms, 01011100=17.6 ms, 01100000=19.2 ms, 01100100=20.8 ms, 01101000=22.4 ms, 01101100=24.0 ms, 01110000=25.6 ms
           TBEN_L4_8IOL:C.Data[36].2   // IO-Link Port 2 - Cycle time (ENUM bit2): 01110100=27.2 ms, 01111000=28.8 ms, 01111100=30.4 ms, 10000000=32.0 ms, 10000001=33.6 ms, 10000010=35.2 ms, 10000011=36.8 ms, 10000100=38.4 ms, 10000101=40.0 ms, 10000110=41.6 ms, 10000111=43.2 ms, 10001000=44.8 ms
           TBEN_L4_8IOL:C.Data[36].3   // IO-Link Port 2 - Cycle time (ENUM bit3): 10001001=46.4 ms, 10001010=48.0 ms, 10001011=49.6 ms, 10001100=51.2 ms, 10001101=52.8 ms, 10001110=54.4 ms, 10001111=56.0 ms, 10010000=57.6 ms, 10010001=59.2 ms, 10010010=60.8 ms, 10010011=62.4 ms, 10010100=64.0 ms
           TBEN_L4_8IOL:C.Data[36].4   // IO-Link Port 2 - Cycle time (ENUM bit4): 10010101=65.6 ms, 10010110=67.2 ms, 10010111=68.8 ms, 10011000=70.4 ms, 10011001=72.0 ms, 10011010=73.6 ms, 10011011=75.2 ms, 10011100=76.8 ms, 10011101=78.4 ms, 10011110=80.0 ms, 10011111=81.6 ms
           TBEN_L4_8IOL:C.Data[36].5   // IO-Link Port 2 - Cycle time (ENUM bit5): 10100000=83.2 ms, 10100001=84.8 ms, 10100010=86.4 ms, 10100011=88.0 ms, 10100100=89.6 ms, 10100101=91.2 ms, 10100110=92.8 ms, 10100111=94.4 ms, 10101000=96.0 ms, 10101001=97.6 ms, 10101010=99.2 ms
           TBEN_L4_8IOL:C.Data[36].6   // IO-Link Port 2 - Cycle time (ENUM bit6): 10101011=100.8 ms, 10101100=102.4 ms, 10101101=104.0 ms, 10101110=105.6 ms, 10101111=107.2 ms, 10110000=108.8 ms, 10110001=110.4 ms, 10110010=112.0 ms, 10110011=113.6 ms, 10110100=115.2 ms, 10110101=116.8 ms
           TBEN_L4_8IOL:C.Data[36].7   // IO-Link Port 2 - Cycle time (ENUM bit7): 10110110=118.4 ms, 10110111=120.0 ms, 10111000=121.6 ms, 10111001=123.2 ms, 10111010=124.8 ms, 10111011=126.4 ms, 10111100=128.0 ms, 10111101=129.6 ms, 10111110=131.2 ms, 10111111=132.8 ms, 11111111=automatic, compatible
           TBEN_L4_8IOL:C.Data[37]   // IO-Link Port 2 - Revision
           TBEN_L4_8IOL:C.Data[37].0   // IO-Link Port 2 - Revision (ENUM bit0): 0=automatic, 1=V1.0
           TBEN_L4_8IOL:C.Data[37].1   // Reserved
           TBEN_L4_8IOL:C.Data[37].2   // Reserved
           TBEN_L4_8IOL:C.Data[37].3   // Reserved
           TBEN_L4_8IOL:C.Data[37].4   // Reserved
           TBEN_L4_8IOL:C.Data[37].5   // Reserved
           TBEN_L4_8IOL:C.Data[37].6   // Reserved
           TBEN_L4_8IOL:C.Data[37].7   // Reserved
           TBEN_L4_8IOL:C.Data[38]   // IO-Link Port 2 - Activate Quick Start-Up
           TBEN_L4_8IOL:C.Data[38].0   // IO-Link Port 2 - Activate Quick Start-Up (ENUM bit0): 0=no, 1=yes
           TBEN_L4_8IOL:C.Data[38].1   // Reserved
           TBEN_L4_8IOL:C.Data[38].2   // Reserved
           TBEN_L4_8IOL:C.Data[38].3   // Reserved
           TBEN_L4_8IOL:C.Data[38].4   // Reserved
           TBEN_L4_8IOL:C.Data[38].5   // Reserved
           TBEN_L4_8IOL:C.Data[38].6   // Reserved
           TBEN_L4_8IOL:C.Data[38].7   // Reserved
           TBEN_L4_8IOL:C.Data[39]   // IO-Link Port 2 - Device parametrization via GSD
           TBEN_L4_8IOL:C.Data[39].0   // IO-Link Port 2 - Device parametrization via GSD (ENUM bit0): 0=inactive, 1=active
           TBEN_L4_8IOL:C.Data[39].1   // Reserved
           TBEN_L4_8IOL:C.Data[39].2   // Reserved
           TBEN_L4_8IOL:C.Data[39].3   // Reserved
           TBEN_L4_8IOL:C.Data[39].4   // Reserved
           TBEN_L4_8IOL:C.Data[39].5   // Reserved
           TBEN_L4_8IOL:C.Data[39].6   // Reserved
           TBEN_L4_8IOL:C.Data[39].7   // Reserved
           TBEN_L4_8IOL:C.Data[40]   // IO-Link Port 2 - Process input data invalid
           TBEN_L4_8IOL:C.Data[40].0   // IO-Link Port 2 - Process input data invalid (ENUM bit0): 0=diagnostic generated, 1=no diagnostic generated
           TBEN_L4_8IOL:C.Data[40].1   // Reserved
           TBEN_L4_8IOL:C.Data[40].2   // Reserved
           TBEN_L4_8IOL:C.Data[40].3   // Reserved
           TBEN_L4_8IOL:C.Data[40].4   // Reserved
           TBEN_L4_8IOL:C.Data[40].5   // Reserved
           TBEN_L4_8IOL:C.Data[40].6   // Reserved
           TBEN_L4_8IOL:C.Data[40].7   // Reserved
           TBEN_L4_8IOL:C.Data[41]   // IO-Link Port 2 - Deactivate diagnostics
           TBEN_L4_8IOL:C.Data[41].0   // IO-Link Port 2 - Deactivate diagnostics (ENUM bit0): 00=no, 01=notifications
           TBEN_L4_8IOL:C.Data[41].1   // IO-Link Port 2 - Deactivate diagnostics (ENUM bit1): 10=notifications and warnings, 11=yes
           TBEN_L4_8IOL:C.Data[41].2   // Reserved
           TBEN_L4_8IOL:C.Data[41].3   // Reserved
           TBEN_L4_8IOL:C.Data[41].4   // Reserved
           TBEN_L4_8IOL:C.Data[41].5   // Reserved
           TBEN_L4_8IOL:C.Data[41].6   // Reserved
           TBEN_L4_8IOL:C.Data[41].7   // Reserved
           TBEN_L4_8IOL:C.Data[42]   // IO-Link Port 2 - Input data mapping
           TBEN_L4_8IOL:C.Data[42].0   // IO-Link Port 2 - Input data mapping (ENUM bit0): 00=direct, 01=swap 16 bit
           TBEN_L4_8IOL:C.Data[42].1   // IO-Link Port 2 - Input data mapping (ENUM bit1): 10=swap 32 bit, 11=swap
           TBEN_L4_8IOL:C.Data[42].2   // Reserved
           TBEN_L4_8IOL:C.Data[42].3   // Reserved
           TBEN_L4_8IOL:C.Data[42].4   // Reserved
           TBEN_L4_8IOL:C.Data[42].5   // Reserved
           TBEN_L4_8IOL:C.Data[42].6   // Reserved
           TBEN_L4_8IOL:C.Data[42].7   // Reserved
           TBEN_L4_8IOL:C.Data[43]   // IO-Link Port 2 - Output data mapping
           TBEN_L4_8IOL:C.Data[43].0   // IO-Link Port 2 - Output data mapping (ENUM bit0): 00=direct, 01=swap 16 bit
           TBEN_L4_8IOL:C.Data[43].1   // IO-Link Port 2 - Output data mapping (ENUM bit1): 10=swap 32 bit, 11=swap
           TBEN_L4_8IOL:C.Data[43].2   // Reserved
           TBEN_L4_8IOL:C.Data[43].3   // Reserved
           TBEN_L4_8IOL:C.Data[43].4   // Reserved
           TBEN_L4_8IOL:C.Data[43].5   // Reserved
           TBEN_L4_8IOL:C.Data[43].6   // Reserved
           TBEN_L4_8IOL:C.Data[43].7   // Reserved
           TBEN_L4_8IOL:C.Data[44]   // IO-Link Port 2 - Vendor ID
           TBEN_L4_8IOL:C.Data[44].0   // IO-Link Port 2 - Vendor ID (INT bit0)
           TBEN_L4_8IOL:C.Data[44].1   // IO-Link Port 2 - Vendor ID (INT bit1)
           TBEN_L4_8IOL:C.Data[44].2   // IO-Link Port 2 - Vendor ID (INT bit2)
           TBEN_L4_8IOL:C.Data[44].3   // IO-Link Port 2 - Vendor ID (INT bit3)
           TBEN_L4_8IOL:C.Data[44].4   // IO-Link Port 2 - Vendor ID (INT bit4)
           TBEN_L4_8IOL:C.Data[44].5   // IO-Link Port 2 - Vendor ID (INT bit5)
           TBEN_L4_8IOL:C.Data[44].6   // IO-Link Port 2 - Vendor ID (INT bit6)
           TBEN_L4_8IOL:C.Data[44].7   // IO-Link Port 2 - Vendor ID (INT bit7)
           TBEN_L4_8IOL:C.Data[45]   // IO-Link Port 2 - Vendor ID
           TBEN_L4_8IOL:C.Data[45].0   // IO-Link Port 2 - Vendor ID (INT bit8)
           TBEN_L4_8IOL:C.Data[45].1   // IO-Link Port 2 - Vendor ID (INT bit9)
           TBEN_L4_8IOL:C.Data[45].2   // IO-Link Port 2 - Vendor ID (INT bit10)
           TBEN_L4_8IOL:C.Data[45].3   // IO-Link Port 2 - Vendor ID (INT bit11)
           TBEN_L4_8IOL:C.Data[45].4   // IO-Link Port 2 - Vendor ID (INT bit12)
           TBEN_L4_8IOL:C.Data[45].5   // IO-Link Port 2 - Vendor ID (INT bit13)
           TBEN_L4_8IOL:C.Data[45].6   // IO-Link Port 2 - Vendor ID (INT bit14)
           TBEN_L4_8IOL:C.Data[45].7   // IO-Link Port 2 - Vendor ID (INT bit15)
           TBEN_L4_8IOL:C.Data[46]   // IO-Link Port 2 - Device ID
           TBEN_L4_8IOL:C.Data[46].0   // IO-Link Port 2 - Device ID (INT bit0)
           TBEN_L4_8IOL:C.Data[46].1   // IO-Link Port 2 - Device ID (INT bit1)
           TBEN_L4_8IOL:C.Data[46].2   // IO-Link Port 2 - Device ID (INT bit2)
           TBEN_L4_8IOL:C.Data[46].3   // IO-Link Port 2 - Device ID (INT bit3)
           TBEN_L4_8IOL:C.Data[46].4   // IO-Link Port 2 - Device ID (INT bit4)
           TBEN_L4_8IOL:C.Data[46].5   // IO-Link Port 2 - Device ID (INT bit5)
           TBEN_L4_8IOL:C.Data[46].6   // IO-Link Port 2 - Device ID (INT bit6)
           TBEN_L4_8IOL:C.Data[46].7   // IO-Link Port 2 - Device ID (INT bit7)
           TBEN_L4_8IOL:C.Data[47]   // IO-Link Port 2 - Device ID
           TBEN_L4_8IOL:C.Data[47].0   // IO-Link Port 2 - Device ID (INT bit8)
           TBEN_L4_8IOL:C.Data[47].1   // IO-Link Port 2 - Device ID (INT bit9)
           TBEN_L4_8IOL:C.Data[47].2   // IO-Link Port 2 - Device ID (INT bit10)
           TBEN_L4_8IOL:C.Data[47].3   // IO-Link Port 2 - Device ID (INT bit11)
           TBEN_L4_8IOL:C.Data[47].4   // IO-Link Port 2 - Device ID (INT bit12)
           TBEN_L4_8IOL:C.Data[47].5   // IO-Link Port 2 - Device ID (INT bit13)
           TBEN_L4_8IOL:C.Data[47].6   // IO-Link Port 2 - Device ID (INT bit14)
           TBEN_L4_8IOL:C.Data[47].7   // IO-Link Port 2 - Device ID (INT bit15)
           TBEN_L4_8IOL:C.Data[48]   // IO-Link Port 2 - Device ID
           TBEN_L4_8IOL:C.Data[48].0   // IO-Link Port 2 - Device ID (INT bit16)
           TBEN_L4_8IOL:C.Data[48].1   // IO-Link Port 2 - Device ID (INT bit17)
           TBEN_L4_8IOL:C.Data[48].2   // IO-Link Port 2 - Device ID (INT bit18)
           TBEN_L4_8IOL:C.Data[48].3   // IO-Link Port 2 - Device ID (INT bit19)
           TBEN_L4_8IOL:C.Data[48].4   // IO-Link Port 2 - Device ID (INT bit20)
           TBEN_L4_8IOL:C.Data[48].5   // IO-Link Port 2 - Device ID (INT bit21)
           TBEN_L4_8IOL:C.Data[48].6   // IO-Link Port 2 - Device ID (INT bit22)
           TBEN_L4_8IOL:C.Data[48].7   // IO-Link Port 2 - Device ID (INT bit23)
           TBEN_L4_8IOL:C.Data[49]   // IO-Link Port 2 - Device ID
           TBEN_L4_8IOL:C.Data[49].0   // IO-Link Port 2 - Device ID (INT bit24)
           TBEN_L4_8IOL:C.Data[49].1   // IO-Link Port 2 - Device ID (INT bit25)
           TBEN_L4_8IOL:C.Data[49].2   // IO-Link Port 2 - Device ID (INT bit26)
           TBEN_L4_8IOL:C.Data[49].3   // IO-Link Port 2 - Device ID (INT bit27)
           TBEN_L4_8IOL:C.Data[49].4   // IO-Link Port 2 - Device ID (INT bit28)
           TBEN_L4_8IOL:C.Data[49].5   // IO-Link Port 2 - Device ID (INT bit29)
           TBEN_L4_8IOL:C.Data[49].6   // IO-Link Port 2 - Device ID (INT bit30)
           TBEN_L4_8IOL:C.Data[49].7   // IO-Link Port 2 - Device ID (INT bit31)
           TBEN_L4_8IOL:C.Data[50]   // IO-Link Port 3 - Operation mode
           TBEN_L4_8IOL:C.Data[50].0   // IO-Link Port 3 - Operation mode (ENUM bit0): 0000=IO-Link without validation, 0001=IO-Link with family compatible device
           TBEN_L4_8IOL:C.Data[50].1   // IO-Link Port 3 - Operation mode (ENUM bit1): 0010=IO-Link with compatible device, 0011=IO-Link with identical device
           TBEN_L4_8IOL:C.Data[50].2   // IO-Link Port 3 - Operation mode (ENUM bit2): 0100=DI (with parameter access)
           TBEN_L4_8IOL:C.Data[50].3   // IO-Link Port 3 - Operation mode (ENUM bit3): 1000=DI
           TBEN_L4_8IOL:C.Data[50].4   // Reserved
           TBEN_L4_8IOL:C.Data[50].5   // Reserved
           TBEN_L4_8IOL:C.Data[50].6   // Reserved
           TBEN_L4_8IOL:C.Data[50].7   // Reserved
           TBEN_L4_8IOL:C.Data[51]   // IO-Link Port 3 - Data storage mode
           TBEN_L4_8IOL:C.Data[51].0   // IO-Link Port 3 - Data storage mode (ENUM bit0): 00=activated, 01=overwrite
           TBEN_L4_8IOL:C.Data[51].1   // IO-Link Port 3 - Data storage mode (ENUM bit1): 10=read in, 11=deactivated, clear
           TBEN_L4_8IOL:C.Data[51].2   // Reserved
           TBEN_L4_8IOL:C.Data[51].3   // Reserved
           TBEN_L4_8IOL:C.Data[51].4   // Reserved
           TBEN_L4_8IOL:C.Data[51].5   // Reserved
           TBEN_L4_8IOL:C.Data[51].6   // Reserved
           TBEN_L4_8IOL:C.Data[51].7   // Reserved
           TBEN_L4_8IOL:C.Data[52]   // IO-Link Port 3 - Cycle time
           TBEN_L4_8IOL:C.Data[52].0   // IO-Link Port 3 - Cycle time (ENUM bit0): 00000000=automatic, 00010000=1.6 ms, 00011000=2.4 ms, 00100000=3.2 ms, 00101000=4.0 ms, 00110000=4.8 ms, 00111000=5.6 ms, 01000000=6.4 ms, 01000010=7.2 ms, 01000100=8.0 ms, 01000110=8.8 ms, 01001000=9.6 ms
           TBEN_L4_8IOL:C.Data[52].1   // IO-Link Port 3 - Cycle time (ENUM bit1): 01001010=10.4 ms, 01001100=11.2 ms, 01001110=12.0 ms, 01010000=12.8 ms, 01010100=14.4 ms, 01011000=16.0 ms, 01011100=17.6 ms, 01100000=19.2 ms, 01100100=20.8 ms, 01101000=22.4 ms, 01101100=24.0 ms, 01110000=25.6 ms
           TBEN_L4_8IOL:C.Data[52].2   // IO-Link Port 3 - Cycle time (ENUM bit2): 01110100=27.2 ms, 01111000=28.8 ms, 01111100=30.4 ms, 10000000=32.0 ms, 10000001=33.6 ms, 10000010=35.2 ms, 10000011=36.8 ms, 10000100=38.4 ms, 10000101=40.0 ms, 10000110=41.6 ms, 10000111=43.2 ms, 10001000=44.8 ms
           TBEN_L4_8IOL:C.Data[52].3   // IO-Link Port 3 - Cycle time (ENUM bit3): 10001001=46.4 ms, 10001010=48.0 ms, 10001011=49.6 ms, 10001100=51.2 ms, 10001101=52.8 ms, 10001110=54.4 ms, 10001111=56.0 ms, 10010000=57.6 ms, 10010001=59.2 ms, 10010010=60.8 ms, 10010011=62.4 ms, 10010100=64.0 ms
           TBEN_L4_8IOL:C.Data[52].4   // IO-Link Port 3 - Cycle time (ENUM bit4): 10010101=65.6 ms, 10010110=67.2 ms, 10010111=68.8 ms, 10011000=70.4 ms, 10011001=72.0 ms, 10011010=73.6 ms, 10011011=75.2 ms, 10011100=76.8 ms, 10011101=78.4 ms, 10011110=80.0 ms, 10011111=81.6 ms
           TBEN_L4_8IOL:C.Data[52].5   // IO-Link Port 3 - Cycle time (ENUM bit5): 10100000=83.2 ms, 10100001=84.8 ms, 10100010=86.4 ms, 10100011=88.0 ms, 10100100=89.6 ms, 10100101=91.2 ms, 10100110=92.8 ms, 10100111=94.4 ms, 10101000=96.0 ms, 10101001=97.6 ms, 10101010=99.2 ms
           TBEN_L4_8IOL:C.Data[52].6   // IO-Link Port 3 - Cycle time (ENUM bit6): 10101011=100.8 ms, 10101100=102.4 ms, 10101101=104.0 ms, 10101110=105.6 ms, 10101111=107.2 ms, 10110000=108.8 ms, 10110001=110.4 ms, 10110010=112.0 ms, 10110011=113.6 ms, 10110100=115.2 ms, 10110101=116.8 ms
           TBEN_L4_8IOL:C.Data[52].7   // IO-Link Port 3 - Cycle time (ENUM bit7): 10110110=118.4 ms, 10110111=120.0 ms, 10111000=121.6 ms, 10111001=123.2 ms, 10111010=124.8 ms, 10111011=126.4 ms, 10111100=128.0 ms, 10111101=129.6 ms, 10111110=131.2 ms, 10111111=132.8 ms, 11111111=automatic, compatible
           TBEN_L4_8IOL:C.Data[53]   // IO-Link Port 3 - Revision
           TBEN_L4_8IOL:C.Data[53].0   // IO-Link Port 3 - Revision (ENUM bit0): 0=automatic, 1=V1.0
           TBEN_L4_8IOL:C.Data[53].1   // Reserved
           TBEN_L4_8IOL:C.Data[53].2   // Reserved
           TBEN_L4_8IOL:C.Data[53].3   // Reserved
           TBEN_L4_8IOL:C.Data[53].4   // Reserved
           TBEN_L4_8IOL:C.Data[53].5   // Reserved
           TBEN_L4_8IOL:C.Data[53].6   // Reserved
           TBEN_L4_8IOL:C.Data[53].7   // Reserved
           TBEN_L4_8IOL:C.Data[54]   // IO-Link Port 3 - Activate Quick Start-Up
           TBEN_L4_8IOL:C.Data[54].0   // IO-Link Port 3 - Activate Quick Start-Up (ENUM bit0): 0=no, 1=yes
           TBEN_L4_8IOL:C.Data[54].1   // Reserved
           TBEN_L4_8IOL:C.Data[54].2   // Reserved
           TBEN_L4_8IOL:C.Data[54].3   // Reserved
           TBEN_L4_8IOL:C.Data[54].4   // Reserved
           TBEN_L4_8IOL:C.Data[54].5   // Reserved
           TBEN_L4_8IOL:C.Data[54].6   // Reserved
           TBEN_L4_8IOL:C.Data[54].7   // Reserved
           TBEN_L4_8IOL:C.Data[55]   // IO-Link Port 3 - Device parametrization via GSD
           TBEN_L4_8IOL:C.Data[55].0   // IO-Link Port 3 - Device parametrization via GSD (ENUM bit0): 0=inactive, 1=active
           TBEN_L4_8IOL:C.Data[55].1   // Reserved
           TBEN_L4_8IOL:C.Data[55].2   // Reserved
           TBEN_L4_8IOL:C.Data[55].3   // Reserved
           TBEN_L4_8IOL:C.Data[55].4   // Reserved
           TBEN_L4_8IOL:C.Data[55].5   // Reserved
           TBEN_L4_8IOL:C.Data[55].6   // Reserved
           TBEN_L4_8IOL:C.Data[55].7   // Reserved
           TBEN_L4_8IOL:C.Data[56]   // IO-Link Port 3 - Process input data invalid
           TBEN_L4_8IOL:C.Data[56].0   // IO-Link Port 3 - Process input data invalid (ENUM bit0): 0=diagnostic generated, 1=no diagnostic generated
           TBEN_L4_8IOL:C.Data[56].1   // Reserved
           TBEN_L4_8IOL:C.Data[56].2   // Reserved
           TBEN_L4_8IOL:C.Data[56].3   // Reserved
           TBEN_L4_8IOL:C.Data[56].4   // Reserved
           TBEN_L4_8IOL:C.Data[56].5   // Reserved
           TBEN_L4_8IOL:C.Data[56].6   // Reserved
           TBEN_L4_8IOL:C.Data[56].7   // Reserved
           TBEN_L4_8IOL:C.Data[57]   // IO-Link Port 3 - Deactivate diagnostics
           TBEN_L4_8IOL:C.Data[57].0   // IO-Link Port 3 - Deactivate diagnostics (ENUM bit0): 00=no, 01=notifications
           TBEN_L4_8IOL:C.Data[57].1   // IO-Link Port 3 - Deactivate diagnostics (ENUM bit1): 10=notifications and warnings, 11=yes
           TBEN_L4_8IOL:C.Data[57].2   // Reserved
           TBEN_L4_8IOL:C.Data[57].3   // Reserved
           TBEN_L4_8IOL:C.Data[57].4   // Reserved
           TBEN_L4_8IOL:C.Data[57].5   // Reserved
           TBEN_L4_8IOL:C.Data[57].6   // Reserved
           TBEN_L4_8IOL:C.Data[57].7   // Reserved
           TBEN_L4_8IOL:C.Data[58]   // IO-Link Port 3 - Input data mapping
           TBEN_L4_8IOL:C.Data[58].0   // IO-Link Port 3 - Input data mapping (ENUM bit0): 00=direct, 01=swap 16 bit
           TBEN_L4_8IOL:C.Data[58].1   // IO-Link Port 3 - Input data mapping (ENUM bit1): 10=swap 32 bit, 11=swap
           TBEN_L4_8IOL:C.Data[58].2   // Reserved
           TBEN_L4_8IOL:C.Data[58].3   // Reserved
           TBEN_L4_8IOL:C.Data[58].4   // Reserved
           TBEN_L4_8IOL:C.Data[58].5   // Reserved
           TBEN_L4_8IOL:C.Data[58].6   // Reserved
           TBEN_L4_8IOL:C.Data[58].7   // Reserved
